// TIA Portal project "openness_project_20230906_002120" (V17)

(* hardware
DEVICE "n0001-zp001-el001-k30001"  S7-1500 station
   slot 0: "Rail_0"  Rack  6ES7 590-1***0-0AA0
   slot 1: "n0001-zp001-el001-k30001"  CPU 1517F-3 PN/DP  6ES7 517-3FP00-0AB0  V2.9
      slot 3: "CPU display_1"  6ES7591-1BA00-0AA0
      slot 32768: "PROFINET interface_1"  X1
         slot 32769: "Port_1"  X1 P1
         slot 32770: "Port_2"  X1 P2
      slot 33024: "PROFINET interface_2"  X2
         slot 33025: "Port_1"  X2 P1
      slot 33280: "DP interface_1"  X3
      slot 34817: "Virtual CP interface port_1"  Virtual CP interface port  Virtual CP interface port
   slot 2: "n0001-zp001-el001-k30002"  CM 1542-1  6GK7 542-1AX00-0XE0  V3.0
DEVICE "n0006-zp001-el001-k25501"  PnPn.Device
   slot 0: "Rack"  Rail  1.0
   slot 0: "n0006-zp001-el001-k25501"  PN/PN Coupler  6ES7 158-3AD10-0XA0  V4.2
   slot 1: "SC01-SORTER-UCOY"  PN/PN Coupler  6ES7 158-3AD10-0XA0  V4.2
   slot 127: "BA 2xRJ45"  BA 2xRJ45  6ES7 193-6AR00-0AA0  V0.0
      slot 1: "Port_1"  X1 P1 R  6ES7 193-6AR00-0AA0  V0.0
      slot 2: "Port_2"  X1 P2 R  6ES7 193-6AR00-0AA0  V0.0
   slot 127: "BA 2xRJ45"  BA 2xRJ45  6ES7 193-6AR00-0AA0  V0.0
      slot 1: "Port_1"  X2 P1 R  6ES7 193-6AR00-0AA0  V0.0
      slot 2: "Port_2"  X2 P2 R  6ES7 193-6AR00-0AA0  V0.0
DEVICE "n0007-zp001-el001-k25502"  PnPn.Device
   slot 0: "Rack"  Rail  1.0
   slot 0: "n0007-zp001-el001-k25502"  PN/PN Coupler  6ES7 158-3AD10-0XA0  V4.2
   slot 1: "SC02-SORTER-LCOY"  PN/PN Coupler  6ES7 158-3AD10-0XA0  V4.2
   slot 127: "BA 2xRJ45"  BA 2xRJ45  6ES7 193-6AR00-0AA0  V0.0
      slot 1: "Port_1"  X1 P1 R  6ES7 193-6AR00-0AA0  V0.0
      slot 2: "Port_2"  X1 P2 R  6ES7 193-6AR00-0AA0  V0.0
   slot 127: "BA 2xRJ45"  BA 2xRJ45  6ES7 193-6AR00-0AA0  V0.0
      slot 1: "Port_1"  X2 P1 R  6ES7 193-6AR00-0AA0  V0.0
      slot 2: "Port_2"  X2 P2 R  6ES7 193-6AR00-0AA0  V0.0
DEVICE "n0008-zp001-el001-k25601"  PnPn.Device
   slot 0: "Rack"  Rail  1.0
   slot 0: "n0008-zp001-el001-k25601"  PN/PN Coupler  6ES7 158-3AD10-0XA0  V4.2
   slot 1: "SF03-SORTER-UFLY"  PN/PN Coupler  6ES7 158-3AD10-0XA0  V4.2
   slot 127: "BA 2xRJ45"  BA 2xRJ45  6ES7 193-6AR00-0AA0  V0.0
      slot 1: "Port_1"  X1 P1 R  6ES7 193-6AR00-0AA0  V0.0
      slot 2: "Port_2"  X1 P2 R  6ES7 193-6AR00-0AA0  V0.0
   slot 127: "BA 2xRJ45"  BA 2xRJ45  6ES7 193-6AR00-0AA0  V0.0
      slot 1: "Port_1"  X2 P1 R  6ES7 193-6AR00-0AA0  V0.0
      slot 2: "Port_2"  X2 P2 R  6ES7 193-6AR00-0AA0  V0.0
DEVICE "n0009-zp001-el001-k25602"  PnPn.Device
   slot 0: "Rack"  Rail  1.0
   slot 0: "n0009-zp001-el001-k25602"  PN/PN Coupler  6ES7 158-3AD10-0XA0  V4.2
   slot 1: "SF04-SORTER-LFLY"  PN/PN Coupler  6ES7 158-3AD10-0XA0  V4.2
   slot 127: "BA 2xRJ45"  BA 2xRJ45  6ES7 193-6AR00-0AA0  V0.0
      slot 1: "Port_1"  X1 P1 R  6ES7 193-6AR00-0AA0  V0.0
      slot 2: "Port_2"  X1 P2 R  6ES7 193-6AR00-0AA0  V0.0
   slot 127: "BA 2xRJ45"  BA 2xRJ45  6ES7 193-6AR00-0AA0  V0.0
      slot 1: "Port_1"  X2 P1 R  6ES7 193-6AR00-0AA0  V0.0
      slot 2: "Port_2"  X2 P2 R  6ES7 193-6AR00-0AA0  V0.0
DEVICE "n0005-zp001-el001-k40001"  ET 200SP-Station
   slot 0: "Rack_0"  Rack  6ES5 710-8MAx1
   slot 0: "n0005-zp001-el001-k40001"  IM 155-6 PN ST  6ES7 155-6AU01-0BN0  V4.2
   slot 1: "-K40002"  DI 16x24VDC ST  6ES7 131-6BH01-0BA0  V0.0
      slot 1: "-K40002"  DI 16x24VDC ST
   slot 2: "-K40003"  DI 16x24VDC ST  6ES7 131-6BH01-0BA0  V0.0
      slot 1: "-K40003"  DI 16x24VDC ST
   slot 3: "-K40004"  DI 16x24VDC ST  6ES7 131-6BH01-0BA0  V0.0
      slot 1: "-K40004"  DI 16x24VDC ST
   slot 4: "-K40005"  DI 16x24VDC ST  6ES7 131-6BH01-0BA0  V0.0
      slot 1: "-K40005"  DI 16x24VDC ST
   slot 5: "-K40006"  DI 16x24VDC ST  6ES7 131-6BH01-0BA0  V0.0
      slot 1: "-K40006"  DI 16x24VDC ST
   slot 6: "-K40007"  DI 16x24VDC ST  6ES7 131-6BH01-0BA0  V0.0
      slot 1: "-K40007"  DI 16x24VDC ST
   slot 7: "-K40008"  DI 16x24VDC ST  6ES7 131-6BH01-0BA0  V0.0
      slot 1: "-K40008"  DI 16x24VDC ST
   slot 8: "-K40009"  DI 16x24VDC ST  6ES7 131-6BH01-0BA0  V0.0
      slot 1: "-K40009"  DI 16x24VDC ST
   slot 9: "-K40010"  DI 16x24VDC ST  6ES7 131-6BH01-0BA0  V0.0
      slot 1: "-K40010"  DI 16x24VDC ST
   slot 10: "-K40011"  DI 16x24VDC ST  6ES7 131-6BH01-0BA0  V0.0
      slot 1: "-K40011"  DI 16x24VDC ST
   slot 11: "-K40012"  DI 16x24VDC ST  6ES7 131-6BH01-0BA0  V0.0
      slot 1: "-K40012"  DI 16x24VDC ST
   slot 12: "-K40013"  DI 16x24VDC ST  6ES7 131-6BH01-0BA0  V0.0
      slot 1: "-K40013"  DI 16x24VDC ST
   slot 13: "-K40014"  DI 16x24VDC ST  6ES7 131-6BH01-0BA0  V0.0
      slot 1: "-K40014"  DI 16x24VDC ST
   slot 14: "-K40015"  DI 16x24VDC ST  6ES7 131-6BH01-0BA0  V0.0
      slot 1: "-K40015"  DI 16x24VDC ST
   slot 15: "-K40016"  DI 16x24VDC ST  6ES7 131-6BH01-0BA0  V0.0
      slot 1: "-K40016"  DI 16x24VDC ST
   slot 16: "-K40017"  DI 16x24VDC ST  6ES7 131-6BH01-0BA0  V0.0
      slot 1: "-K40017"  DI 16x24VDC ST
   slot 17: "-K40018"  DI 16x24VDC ST  6ES7 131-6BH01-0BA0  V0.0
      slot 1: "-K40018"  DI 16x24VDC ST
   slot 18: "-K40019"  F-DI 8x24VDC HF  6ES7 136-6BA00-0CA0  V1.0
      slot 1: "-K40019"  F-DI 8x24VDC HF
   slot 19: "-K40020"  DQ 16x24VDC/0.5A ST  6ES7 132-6BH01-0BA0  V0.0
      slot 1: "-K40020"  DQ 16x24VDC/0.5A ST
   slot 20: "Server module_1"  Server module  6ES7 193-6PA00-0AA0  V1.1
      slot 1: "Server module_1"  Server module
   slot 127: "BA 2xRJ45"  BA 2xRJ45  6ES7 193-6AR00-0AA0  V0.0
      slot 1: "Port_1"  X1 P1 R  6ES7 193-6AR00-0AA0  V0.0
      slot 2: "Port_2"  X1 P2 R  6ES7 193-6AR00-0AA0  V0.0
DEVICE "n0013-uf317-xn10"  GSD.Device.PN
   slot 0: "Rack"  Rack  V1.0
   slot 0: "n0013-uf317-xn10"  55556 MVK-MPNIO F DI16/8  55556
      slot 0: "55556 MVK-MPNIO F DI16/8_1"  55556 MVK-MPNIO F DI16/8
      slot 1: "55556 MVK-MPNIO F DI16/8"  55556 MVK-MPNIO F DI16/8
         slot 1: "Port 1"  Port 1
         slot 2: "Port 2"  Port 2
      slot 1: "Power module_1"  Power module
         slot 0: "Power module"  Power module
   slot 2: "-XN10"  FS Data
      slot 0: "-XN10"  FS Data
DEVICE "n0015-uc16-el001-k30001"  ET 200SP-Station
   slot 0: "Rack_0"  Rack  6ES5 710-8MAx1
   slot 0: "n0015-uc16-el001-k30001"  IM 155-6 PN ST  6ES7 155-6AU01-0BN0  V4.2
   slot 1: "-K30002"  DI 16x24VDC ST  6ES7 131-6BH01-0BA0  V0.0
      slot 1: "-K30002"  DI 16x24VDC ST
   slot 2: "-K30003"  DI 16x24VDC ST  6ES7 131-6BH01-0BA0  V0.0
      slot 1: "-K30003"  DI 16x24VDC ST
   slot 3: "-K30004"  F-DI 8x24VDC HF  6ES7 136-6BA00-0CA0  V1.0
      slot 1: "-K30004"  F-DI 8x24VDC HF
   slot 4: "-K30005"  F-DI 8x24VDC HF  6ES7 136-6BA00-0CA0  V1.0
      slot 1: "-K30005"  F-DI 8x24VDC HF
   slot 5: "-K30006"  F-DI 8x24VDC HF  6ES7 136-6BA00-0CA0  V1.0
      slot 1: "-K30006"  F-DI 8x24VDC HF
   slot 6: "-K30007"  F-DI 8x24VDC HF  6ES7 136-6BA00-0CA0  V1.0
      slot 1: "-K30007"  F-DI 8x24VDC HF
   slot 7: "-K30008"  F-DQ 4x24VDC/2A PM HF  6ES7 136-6DB00-0CA0  V2.0
      slot 1: "-K30008"  F-DQ 4x24VDC/2A PM HF
   slot 8: "-K30009"  F-DQ 4x24VDC/2A PM HF  6ES7 136-6DB00-0CA0  V2.0
      slot 1: "-K30009"  F-DQ 4x24VDC/2A PM HF
   slot 9: "-K30010"  F-DQ 4x24VDC/2A PM HF  6ES7 136-6DB00-0CA0  V2.0
      slot 1: "-K30010"  F-DQ 4x24VDC/2A PM HF
   slot 10: "-K30011"  F-DQ 4x24VDC/2A PM HF  6ES7 136-6DB00-0CA0  V2.0
      slot 1: "-K30011"  F-DQ 4x24VDC/2A PM HF
   slot 11: "-K30012"  F-DQ 4x24VDC/2A PM HF  6ES7 136-6DB00-0CA0  V2.0
      slot 1: "-K30012"  F-DQ 4x24VDC/2A PM HF
   slot 12: "-K30013"  F-DQ 4x24VDC/2A PM HF  6ES7 136-6DB00-0CA0  V2.0
      slot 1: "-K30013"  F-DQ 4x24VDC/2A PM HF
   slot 13: "Server module_1"  Server module  6ES7 193-6PA00-0AA0  V1.1
      slot 1: "Server module_1"  Server module
   slot 127: "BA 2xRJ45"  BA 2xRJ45  6ES7 193-6AR00-0AA0  V0.0
      slot 1: "Port_1"  X1 P1 R  6ES7 193-6AR00-0AA0  V0.0
      slot 2: "Port_2"  X1 P2 R  6ES7 193-6AR00-0AA0  V0.0
DEVICE "n0016-uc164-xn10"  GSD.Device.PN
   slot 0: "Rack"  Rack  V1.0
   slot 0: "n0016-uc164-xn10"  55556 MVK-MPNIO F DI16/8  55556
      slot 0: "55556 MVK-MPNIO F DI16/8_1"  55556 MVK-MPNIO F DI16/8
      slot 1: "55556 MVK-MPNIO F DI16/8"  55556 MVK-MPNIO F DI16/8
         slot 1: "Port 1"  Port 1
         slot 2: "Port 2"  Port 2
      slot 1: "Power module_1"  Power module
         slot 0: "Power module"  Power module
   slot 2: "-XN10"  FS Data
      slot 0: "-XN10"  FS Data
DEVICE "n0017-lv004-el001-k30001"  ET 200SP-Station
   slot 0: "Rack_0"  Rack  6ES5 710-8MAx1
   slot 0: "n0017-lv004-el001-k30001"  IM 155-6 PN ST  6ES7 155-6AU01-0BN0  V4.2
   slot 1: "-K30002"  DI 16x24VDC ST  6ES7 131-6BH01-0BA0  V0.0
      slot 1: "-K30002"  DI 16x24VDC ST
   slot 2: "-K30003"  F-DI 8x24VDC HF  6ES7 136-6BA00-0CA0  V1.0
      slot 1: "-K30003"  F-DI 8x24VDC HF
   slot 3: "-K30004"  F-DI 8x24VDC HF  6ES7 136-6BA00-0CA0  V1.0
      slot 1: "-K30004"  F-DI 8x24VDC HF
   slot 4: "-K30005"  F-DQ 4x24VDC/2A PM HF  6ES7 136-6DB00-0CA0  V2.0
      slot 1: "-K30005"  F-DQ 4x24VDC/2A PM HF
   slot 5: "-K30006"  F-DQ 4x24VDC/2A PM HF  6ES7 136-6DB00-0CA0  V2.0
      slot 1: "-K30006"  F-DQ 4x24VDC/2A PM HF
   slot 6: "Server module_1"  Server module  6ES7 193-6PA00-0AA0  V1.1
      slot 1: "Server module_1"  Server module
   slot 127: "BA 2xRJ45"  BA 2xRJ45  6ES7 193-6AR00-0AA0  V0.0
      slot 1: "Port_1"  X1 P1 R  6ES7 193-6AR00-0AA0  V0.0
      slot 2: "Port_2"  X1 P2 R  6ES7 193-6AR00-0AA0  V0.0
DEVICE "n0018-lv004-el001-k30001"  ET 200SP-Station
   slot 0: "Rack_0"  Rack  6ES5 710-8MAx1
   slot 0: "n0018-lv004-el001-k30001"  IM 155-6 PN ST  6ES7 155-6AU01-0BN0  V4.2
   slot 1: "-K30002"  DI 16x24VDC ST  6ES7 131-6BH01-0BA0  V0.0
      slot 1: "-K30002"  DI 16x24VDC ST
   slot 2: "-K30003"  F-DI 8x24VDC HF  6ES7 136-6BA00-0CA0  V1.0
      slot 1: "-K30003"  F-DI 8x24VDC HF
   slot 3: "-K30004"  F-DI 8x24VDC HF  6ES7 136-6BA00-0CA0  V1.0
      slot 1: "-K30004"  F-DI 8x24VDC HF
   slot 4: "-K30005"  F-DQ 4x24VDC/2A PM HF  6ES7 136-6DB00-0CA0  V2.0
      slot 1: "-K30005"  F-DQ 4x24VDC/2A PM HF
   slot 5: "-K30006"  F-DQ 4x24VDC/2A PM HF  6ES7 136-6DB00-0CA0  V2.0
      slot 1: "-K30006"  F-DQ 4x24VDC/2A PM HF
   slot 6: "Server module_1"  Server module  6ES7 193-6PA00-0AA0  V1.1
      slot 1: "Server module_1"  Server module
   slot 127: "BA 2xRJ45"  BA 2xRJ45  6ES7 193-6AR00-0AA0  V0.0
      slot 1: "Port_1"  X1 P1 R  6ES7 193-6AR00-0AA0  V0.0
      slot 2: "Port_2"  X1 P2 R  6ES7 193-6AR00-0AA0  V0.0
DEVICE "n0020-uc15-el001-k30001"  ET 200SP-Station
   slot 0: "Rack_0"  Rack  6ES5 710-8MAx1
   slot 0: "n0020-uc15-el001-k30001"  IM 155-6 PN ST  6ES7 155-6AU01-0BN0  V4.2
   slot 1: "-K30002"  DI 16x24VDC ST  6ES7 131-6BH01-0BA0  V0.0
      slot 1: "-K30002"  DI 16x24VDC ST
   slot 2: "-K30003"  DI 16x24VDC ST  6ES7 131-6BH01-0BA0  V0.0
      slot 1: "-K30003"  DI 16x24VDC ST
   slot 3: "-K30004"  F-DI 8x24VDC HF  6ES7 136-6BA00-0CA0  V1.0
      slot 1: "-K30004"  F-DI 8x24VDC HF
   slot 4: "-K30005"  F-DI 8x24VDC HF  6ES7 136-6BA00-0CA0  V1.0
      slot 1: "-K30005"  F-DI 8x24VDC HF
   slot 5: "-K30006"  F-DI 8x24VDC HF  6ES7 136-6BA00-0CA0  V1.0
      slot 1: "-K30006"  F-DI 8x24VDC HF
   slot 6: "-K30007"  F-DI 8x24VDC HF  6ES7 136-6BA00-0CA0  V1.0
      slot 1: "-K30007"  F-DI 8x24VDC HF
   slot 7: "-K30008"  F-DQ 4x24VDC/2A PM HF  6ES7 136-6DB00-0CA0  V2.0
      slot 1: "-K30008"  F-DQ 4x24VDC/2A PM HF
   slot 8: "-K30009"  F-DQ 4x24VDC/2A PM HF  6ES7 136-6DB00-0CA0  V2.0
      slot 1: "-K30009"  F-DQ 4x24VDC/2A PM HF
   slot 9: "-K30010"  F-DQ 4x24VDC/2A PM HF  6ES7 136-6DB00-0CA0  V2.0
      slot 1: "-K30010"  F-DQ 4x24VDC/2A PM HF
   slot 10: "-K30011"  F-DQ 4x24VDC/2A PM HF  6ES7 136-6DB00-0CA0  V2.0
      slot 1: "-K30011"  F-DQ 4x24VDC/2A PM HF
   slot 11: "-K30012"  F-DQ 4x24VDC/2A PM HF  6ES7 136-6DB00-0CA0  V2.0
      slot 1: "-K30012"  F-DQ 4x24VDC/2A PM HF
   slot 12: "-K30013"  F-DQ 4x24VDC/2A PM HF  6ES7 136-6DB00-0CA0  V2.0
      slot 1: "-K30013"  F-DQ 4x24VDC/2A PM HF
   slot 13: "Server module_1"  Server module  6ES7 193-6PA00-0AA0  V1.1
      slot 1: "Server module_1"  Server module
   slot 127: "BA 2xRJ45"  BA 2xRJ45  6ES7 193-6AR00-0AA0  V0.0
      slot 1: "Port_1"  X1 P1 R  6ES7 193-6AR00-0AA0  V0.0
      slot 2: "Port_2"  X1 P2 R  6ES7 193-6AR00-0AA0  V0.0
DEVICE "n0023-uc154-xn10"  GSD.Device.PN
   slot 0: "Rack"  Rack  V1.0
   slot 0: "n0023-uc154-xn10"  55556 MVK-MPNIO F DI16/8  55556
      slot 0: "55556 MVK-MPNIO F DI16/8_1"  55556 MVK-MPNIO F DI16/8
      slot 1: "55556 MVK-MPNIO F DI16/8"  55556 MVK-MPNIO F DI16/8
         slot 1: "Port 1"  Port 1
         slot 2: "Port 2"  Port 2
      slot 1: "Power module_1"  Power module
         slot 0: "Power module"  Power module
   slot 2: "-XN10"  FS Data
      slot 0: "-XN10"  FS Data
DEVICE "n0021-icg11-el001-k30001"  ET 200SP-Station
   slot 0: "Rack_0"  Rack  6ES5 710-8MAx1
   slot 0: "n0021-icg11-el001-k30001"  IM 155-6 PN ST  6ES7 155-6AU01-0BN0  V4.2
   slot 1: "-K30002"  DI 16x24VDC ST  6ES7 131-6BH01-0BA0  V0.0
      slot 1: "-K30002"  DI 16x24VDC ST
   slot 2: "-K30003"  F-DI 8x24VDC HF  6ES7 136-6BA00-0CA0  V1.0
      slot 1: "-K30003"  F-DI 8x24VDC HF
   slot 3: "-K30004"  F-DI 8x24VDC HF  6ES7 136-6BA00-0CA0  V1.0
      slot 1: "-K30004"  F-DI 8x24VDC HF
   slot 4: "-K30005"  F-DI 8x24VDC HF  6ES7 136-6BA00-0CA0  V1.0
      slot 1: "-K30005"  F-DI 8x24VDC HF
   slot 5: "-K30006"  F-DI 8x24VDC HF  6ES7 136-6BA00-0CA0  V1.0
      slot 1: "-K30006"  F-DI 8x24VDC HF
   slot 6: "-K30007"  F-DQ 4x24VDC/2A PM HF  6ES7 136-6DB00-0CA0  V2.0
      slot 1: "-K30007"  F-DQ 4x24VDC/2A PM HF
   slot 7: "-K30008"  F-DQ 4x24VDC/2A PM HF  6ES7 136-6DB00-0CA0  V2.0
      slot 1: "-K30008"  F-DQ 4x24VDC/2A PM HF
   slot 8: "-K30009"  F-DQ 4x24VDC/2A PM HF  6ES7 136-6DB00-0CA0  V2.0
      slot 1: "-K30009"  F-DQ 4x24VDC/2A PM HF
   slot 9: "Server module_1"  Server module  6ES7 193-6PA00-0AA0  V1.1
      slot 1: "Server module_1"  Server module
   slot 127: "BA 2xRJ45"  BA 2xRJ45  6ES7 193-6AR00-0AA0  V0.0
      slot 1: "Port_1"  X1 P1 R  6ES7 193-6AR00-0AA0  V0.0
      slot 2: "Port_2"  X1 P2 R  6ES7 193-6AR00-0AA0  V0.0
DEVICE "n0022-icg21-el001-k30001"  ET 200SP-Station
   slot 0: "Rack_0"  Rack  6ES5 710-8MAx1
   slot 0: "n0022-icg21-el001-k30001"  IM 155-6 PN ST  6ES7 155-6AU01-0BN0  V4.2
   slot 1: "-K30002"  DI 16x24VDC ST  6ES7 131-6BH01-0BA0  V0.0
      slot 1: "-K30002"  DI 16x24VDC ST
   slot 2: "-K30003"  F-DI 8x24VDC HF  6ES7 136-6BA00-0CA0  V1.0
      slot 1: "-K30003"  F-DI 8x24VDC HF
   slot 3: "-K30004"  F-DI 8x24VDC HF  6ES7 136-6BA00-0CA0  V1.0
      slot 1: "-K30004"  F-DI 8x24VDC HF
   slot 4: "-K30005"  F-DI 8x24VDC HF  6ES7 136-6BA00-0CA0  V1.0
      slot 1: "-K30005"  F-DI 8x24VDC HF
   slot 5: "-K30006"  F-DI 8x24VDC HF  6ES7 136-6BA00-0CA0  V1.0
      slot 1: "-K30006"  F-DI 8x24VDC HF
   slot 6: "-K30007"  F-DQ 4x24VDC/2A PM HF  6ES7 136-6DB00-0CA0  V2.0
      slot 1: "-K30007"  F-DQ 4x24VDC/2A PM HF
   slot 7: "-K30008"  F-DQ 4x24VDC/2A PM HF  6ES7 136-6DB00-0CA0  V2.0
      slot 1: "-K30008"  F-DQ 4x24VDC/2A PM HF
   slot 8: "-K30009"  F-DQ 4x24VDC/2A PM HF  6ES7 136-6DB00-0CA0  V2.0
      slot 1: "-K30009"  F-DQ 4x24VDC/2A PM HF
   slot 9: "Server module_1"  Server module  6ES7 193-6PA00-0AA0  V1.1
      slot 1: "Server module_1"  Server module
   slot 127: "BA 2xRJ45"  BA 2xRJ45  6ES7 193-6AR00-0AA0  V0.0
      slot 1: "Port_1"  X1 P1 R  6ES7 193-6AR00-0AA0  V0.0
      slot 2: "Port_2"  X1 P2 R  6ES7 193-6AR00-0AA0  V0.0
DEVICE "n0025-uc14-el001-k30001"  ET 200SP-Station
   slot 0: "Rack_0"  Rack  6ES5 710-8MAx1
   slot 0: "n0025-uc14-el001-k30001"  IM 155-6 PN ST  6ES7 155-6AU01-0BN0  V4.2
   slot 1: "-K30002"  DI 16x24VDC ST  6ES7 131-6BH01-0BA0  V0.0
      slot 1: "-K30002"  DI 16x24VDC ST
   slot 2: "-K30003"  DI 16x24VDC ST  6ES7 131-6BH01-0BA0  V0.0
      slot 1: "-K30003"  DI 16x24VDC ST
   slot 3: "-K30004"  F-DI 8x24VDC HF  6ES7 136-6BA00-0CA0  V1.0
      slot 1: "-K30004"  F-DI 8x24VDC HF
   slot 4: "-K30005"  F-DI 8x24VDC HF  6ES7 136-6BA00-0CA0  V1.0
      slot 1: "-K30005"  F-DI 8x24VDC HF
   slot 5: "-K30006"  F-DI 8x24VDC HF  6ES7 136-6BA00-0CA0  V1.0
      slot 1: "-K30006"  F-DI 8x24VDC HF
   slot 6: "-K30007"  F-DI 8x24VDC HF  6ES7 136-6BA00-0CA0  V1.0
      slot 1: "-K30007"  F-DI 8x24VDC HF
   slot 7: "-K30008"  F-DQ 4x24VDC/2A PM HF  6ES7 136-6DB00-0CA0  V2.0
      slot 1: "-K30008"  F-DQ 4x24VDC/2A PM HF
   slot 8: "-K30009"  F-DQ 4x24VDC/2A PM HF  6ES7 136-6DB00-0CA0  V2.0
      slot 1: "-K30009"  F-DQ 4x24VDC/2A PM HF
   slot 9: "-K30010"  F-DQ 4x24VDC/2A PM HF  6ES7 136-6DB00-0CA0  V2.0
      slot 1: "-K30010"  F-DQ 4x24VDC/2A PM HF
   slot 10: "-K30011"  F-DQ 4x24VDC/2A PM HF  6ES7 136-6DB00-0CA0  V2.0
      slot 1: "-K30011"  F-DQ 4x24VDC/2A PM HF
   slot 11: "-K30012"  F-DQ 4x24VDC/2A PM HF  6ES7 136-6DB00-0CA0  V2.0
      slot 1: "-K30012"  F-DQ 4x24VDC/2A PM HF
   slot 12: "-K30013"  F-DQ 4x24VDC/2A PM HF  6ES7 136-6DB00-0CA0  V2.0
      slot 1: "-K30013"  F-DQ 4x24VDC/2A PM HF
   slot 13: "Server module_1"  Server module  6ES7 193-6PA00-0AA0  V1.1
      slot 1: "Server module_1"  Server module
   slot 127: "BA 2xRJ45"  BA 2xRJ45  6ES7 193-6AR00-0AA0  V0.0
      slot 1: "Port_1"  X1 P1 R  6ES7 193-6AR00-0AA0  V0.0
      slot 2: "Port_2"  X1 P2 R  6ES7 193-6AR00-0AA0  V0.0
DEVICE "n0026-uc144-xn10"  GSD.Device.PN
   slot 0: "Rack"  Rack  V1.0
   slot 0: "n0026-uc144-xn10"  55556 MVK-MPNIO F DI16/8  55556
      slot 0: "55556 MVK-MPNIO F DI16/8_1"  55556 MVK-MPNIO F DI16/8
      slot 1: "55556 MVK-MPNIO F DI16/8"  55556 MVK-MPNIO F DI16/8
         slot 1: "Port 1"  Port 1
         slot 2: "Port 2"  Port 2
      slot 1: "Power module_1"  Power module
         slot 0: "Power module"  Power module
   slot 2: "-XN10"  FS Data
      slot 0: "-XN10"  FS Data
DEVICE "n0038-uc1-el001-k30001"  ET 200SP-Station
   slot 0: "Rack_0"  Rack  6ES5 710-8MAx1
   slot 0: "n0038-uc1-el001-k30001"  IM 155-6 PN ST  6ES7 155-6AU01-0BN0  V4.2
   slot 1: "-K30002"  DI 16x24VDC ST  6ES7 131-6BH01-0BA0  V0.0
      slot 1: "-K30002"  DI 16x24VDC ST
   slot 2: "-K30003"  F-DI 8x24VDC HF  6ES7 136-6BA00-0CA0  V1.0
      slot 1: "-K30003"  F-DI 8x24VDC HF
   slot 3: "-K30004"  F-DI 8x24VDC HF  6ES7 136-6BA00-0CA0  V1.0
      slot 1: "-K30004"  F-DI 8x24VDC HF
   slot 4: "-K30005"  F-DQ 4x24VDC/2A PM HF  6ES7 136-6DB00-0CA0  V2.0
      slot 1: "-K30005"  F-DQ 4x24VDC/2A PM HF
   slot 5: "-K30006"  DQ 16x24VDC/0.5A ST  6ES7 132-6BH01-0BA0  V0.0
      slot 1: "-K30006"  DQ 16x24VDC/0.5A ST
   slot 6: "Server module_1"  Server module  6ES7 193-6PA00-0AA0  V1.1
      slot 1: "Server module_1"  Server module
   slot 127: "BA 2xRJ45"  BA 2xRJ45  6ES7 193-6AR00-0AA0  V0.0
      slot 1: "Port_1"  X1 P1 R  6ES7 193-6AR00-0AA0  V0.0
      slot 2: "Port_2"  X1 P2 R  6ES7 193-6AR00-0AA0  V0.0
DEVICE "n0039-lv001-el001-k30001"  ET 200SP-Station
   slot 0: "Rack_0"  Rack  6ES5 710-8MAx1
   slot 0: "n0039-lv001-el001-k30001"  IM 155-6 PN ST  6ES7 155-6AU01-0BN0  V4.2
   slot 1: "-K30002"  DI 16x24VDC ST  6ES7 131-6BH01-0BA0  V0.0
      slot 1: "-K30002"  DI 16x24VDC ST
   slot 2: "-K30003"  F-DI 8x24VDC HF  6ES7 136-6BA00-0CA0  V1.0
      slot 1: "-K30003"  F-DI 8x24VDC HF
   slot 3: "-K30004"  F-DQ 4x24VDC/2A PM HF  6ES7 136-6DB00-0CA0  V2.0
      slot 1: "-K30004"  F-DQ 4x24VDC/2A PM HF
   slot 4: "Server module_1"  Server module  6ES7 193-6PA00-0AA0  V1.1
      slot 1: "Server module_1"  Server module
   slot 127: "BA 2xRJ45"  BA 2xRJ45  6ES7 193-6AR00-0AA0  V0.0
      slot 1: "Port_1"  X1 P1 R  6ES7 193-6AR00-0AA0  V0.0
      slot 2: "Port_2"  X1 P2 R  6ES7 193-6AR00-0AA0  V0.0
DEVICE "n0040-lv001-el001-k30001"  ET 200SP-Station
   slot 0: "Rack_0"  Rack  6ES5 710-8MAx1
   slot 0: "n0040-lv001-el001-k30001"  IM 155-6 PN ST  6ES7 155-6AU01-0BN0  V4.2
   slot 1: "-K30002"  DI 16x24VDC ST  6ES7 131-6BH01-0BA0  V0.0
      slot 1: "-K30002"  DI 16x24VDC ST
   slot 2: "-K30003"  F-DI 8x24VDC HF  6ES7 136-6BA00-0CA0  V1.0
      slot 1: "-K30003"  F-DI 8x24VDC HF
   slot 3: "-K30004"  F-DQ 4x24VDC/2A PM HF  6ES7 136-6DB00-0CA0  V2.0
      slot 1: "-K30004"  F-DQ 4x24VDC/2A PM HF
   slot 4: "Server module_1"  Server module  6ES7 193-6PA00-0AA0  V1.1
      slot 1: "Server module_1"  Server module
   slot 127: "BA 2xRJ45"  BA 2xRJ45  6ES7 193-6AR00-0AA0  V0.0
      slot 1: "Port_1"  X1 P1 R  6ES7 193-6AR00-0AA0  V0.0
      slot 2: "Port_2"  X1 P2 R  6ES7 193-6AR00-0AA0  V0.0
DEVICE "n0041-uf31-el002-k30001"  ET 200SP-Station
   slot 0: "Rack_0"  Rack  6ES5 710-8MAx1
   slot 0: "n0041-uf31-el002-k30001"  IM 155-6 PN ST  6ES7 155-6AU01-0BN0  V4.2
   slot 1: "-K30002"  DI 16x24VDC ST  6ES7 131-6BH01-0BA0  V0.0
      slot 1: "-K30002"  DI 16x24VDC ST
   slot 2: "-K30003"  F-DI 8x24VDC HF  6ES7 136-6BA00-0CA0  V1.0
      slot 1: "-K30003"  F-DI 8x24VDC HF
   slot 3: "-K30004"  F-DI 8x24VDC HF  6ES7 136-6BA00-0CA0  V1.0
      slot 1: "-K30004"  F-DI 8x24VDC HF
   slot 4: "-K30005"  F-DQ 4x24VDC/2A PM HF  6ES7 136-6DB00-0CA0  V2.0
      slot 1: "-K30005"  F-DQ 4x24VDC/2A PM HF
   slot 5: "Server module_1"  Server module  6ES7 193-6PA00-0AA0  V1.1
      slot 1: "Server module_1"  Server module
   slot 127: "BA 2xRJ45"  BA 2xRJ45  6ES7 193-6AR00-0AA0  V0.0
      slot 1: "Port_1"  X1 P1 R  6ES7 193-6AR00-0AA0  V0.0
      slot 2: "Port_2"  X1 P2 R  6ES7 193-6AR00-0AA0  V0.0
DEVICE "n0042-uf41-el002-k30001"  ET 200SP-Station
   slot 0: "Rack_0"  Rack  6ES5 710-8MAx1
   slot 0: "n0042-uf41-el002-k30001"  IM 155-6 PN ST  6ES7 155-6AU01-0BN0  V4.2
   slot 1: "-K30002"  DI 16x24VDC ST  6ES7 131-6BH01-0BA0  V0.0
      slot 1: "-K30002"  DI 16x24VDC ST
   slot 2: "-K30003"  F-DI 8x24VDC HF  6ES7 136-6BA00-0CA0  V1.0
      slot 1: "-K30003"  F-DI 8x24VDC HF
   slot 3: "-K30004"  F-DQ 4x24VDC/2A PM HF  6ES7 136-6DB00-0CA0  V2.0
      slot 1: "-K30004"  F-DQ 4x24VDC/2A PM HF
   slot 4: "-K30005"  F-DQ 4x24VDC/2A PM HF  6ES7 136-6DB00-0CA0  V2.0
      slot 1: "-K30005"  F-DQ 4x24VDC/2A PM HF
   slot 5: "Server module_1"  Server module  6ES7 193-6PA00-0AA0  V1.1
      slot 1: "Server module_1"  Server module
   slot 127: "BA 2xRJ45"  BA 2xRJ45  6ES7 193-6AR00-0AA0  V0.0
      slot 1: "Port_1"  X1 P1 R  6ES7 193-6AR00-0AA0  V0.0
      slot 2: "Port_2"  X1 P2 R  6ES7 193-6AR00-0AA0  V0.0
DEVICE "n0044-ct1-el001-k30001"  ET 200SP-Station
   slot 0: "Rack_0"  Rack  6ES5 710-8MAx1
   slot 0: "n0044-ct1-el001-k30001"  IM 155-6 PN ST  6ES7 155-6AU01-0BN0  V4.2
   slot 1: "-K30002"  DI 16x24VDC ST  6ES7 131-6BH01-0BA0  V0.0
      slot 1: "-K30002"  DI 16x24VDC ST
   slot 2: "-K30003"  F-DI 8x24VDC HF  6ES7 136-6BA00-0CA0  V1.0
      slot 1: "-K30003"  F-DI 8x24VDC HF
   slot 3: "-K30004"  F-DI 8x24VDC HF  6ES7 136-6BA00-0CA0  V1.0
      slot 1: "-K30004"  F-DI 8x24VDC HF
   slot 4: "-K30005"  F-DI 8x24VDC HF  6ES7 136-6BA00-0CA0  V1.0
      slot 1: "-K30005"  F-DI 8x24VDC HF
   slot 5: "-K30006"  F-DI 8x24VDC HF  6ES7 136-6BA00-0CA0  V1.0
      slot 1: "-K30006"  F-DI 8x24VDC HF
   slot 6: "-K30007"  F-DI 8x24VDC HF  6ES7 136-6BA00-0CA0  V1.0
      slot 1: "-K30007"  F-DI 8x24VDC HF
   slot 7: "-K30008"  F-DQ 4x24VDC/2A PM HF  6ES7 136-6DB00-0CA0  V2.0
      slot 1: "-K30008"  F-DQ 4x24VDC/2A PM HF
   slot 8: "-K30009"  F-DQ 4x24VDC/2A PM HF  6ES7 136-6DB00-0CA0  V2.0
      slot 1: "-K30009"  F-DQ 4x24VDC/2A PM HF
   slot 9: "Server module_1"  Server module  6ES7 193-6PA00-0AA0  V1.1
      slot 1: "Server module_1"  Server module
   slot 127: "BA 2xRJ45"  BA 2xRJ45  6ES7 193-6AR00-0AA0  V0.0
      slot 1: "Port_1"  X1 P1 R  6ES7 193-6AR00-0AA0  V0.0
      slot 2: "Port_2"  X1 P2 R  6ES7 193-6AR00-0AA0  V0.0
DEVICE "n0045-ct1-el002-k30001"  ET 200SP-Station
   slot 0: "Rack_0"  Rack  6ES5 710-8MAx1
   slot 0: "n0045-ct1-el002-k30001"  IM 155-6 PN ST  6ES7 155-6AU01-0BN0  V4.2
   slot 1: "-K30002"  DI 16x24VDC ST  6ES7 131-6BH01-0BA0  V0.0
      slot 1: "-K30002"  DI 16x24VDC ST
   slot 2: "-K30003"  F-DI 8x24VDC HF  6ES7 136-6BA00-0CA0  V1.0
      slot 1: "-K30003"  F-DI 8x24VDC HF
   slot 3: "-K30004"  F-DI 8x24VDC HF  6ES7 136-6BA00-0CA0  V1.0
      slot 1: "-K30004"  F-DI 8x24VDC HF
   slot 4: "-K30005"  F-DI 8x24VDC HF  6ES7 136-6BA00-0CA0  V1.0
      slot 1: "-K30005"  F-DI 8x24VDC HF
   slot 5: "-K30006"  F-DI 8x24VDC HF  6ES7 136-6BA00-0CA0  V1.0
      slot 1: "-K30006"  F-DI 8x24VDC HF
   slot 6: "-K30007"  F-DI 8x24VDC HF  6ES7 136-6BA00-0CA0  V1.0
      slot 1: "-K30007"  F-DI 8x24VDC HF
   slot 7: "-K30008"  F-DQ 4x24VDC/2A PM HF  6ES7 136-6DB00-0CA0  V2.0
      slot 1: "-K30008"  F-DQ 4x24VDC/2A PM HF
   slot 8: "-K30009"  F-DQ 4x24VDC/2A PM HF  6ES7 136-6DB00-0CA0  V2.0
      slot 1: "-K30009"  F-DQ 4x24VDC/2A PM HF
   slot 9: "Server module_1"  Server module  6ES7 193-6PA00-0AA0  V1.1
      slot 1: "Server module_1"  Server module
   slot 127: "BA 2xRJ45"  BA 2xRJ45  6ES7 193-6AR00-0AA0  V0.0
      slot 1: "Port_1"  X1 P1 R  6ES7 193-6AR00-0AA0  V0.0
      slot 2: "Port_2"  X1 P2 R  6ES7 193-6AR00-0AA0  V0.0
DEVICE "n0046-ct1-el003-k30001"  ET 200SP-Station
   slot 0: "Rack_0"  Rack  6ES5 710-8MAx1
   slot 0: "n0046-ct1-el003-k30001"  IM 155-6 PN ST  6ES7 155-6AU01-0BN0  V4.2
   slot 1: "-K30002"  DI 16x24VDC ST  6ES7 131-6BH01-0BA0  V0.0
      slot 1: "-K30002"  DI 16x24VDC ST
   slot 2: "-K30003"  F-DI 8x24VDC HF  6ES7 136-6BA00-0CA0  V1.0
      slot 1: "-K30003"  F-DI 8x24VDC HF
   slot 3: "-K30004"  F-DI 8x24VDC HF  6ES7 136-6BA00-0CA0  V1.0
      slot 1: "-K30004"  F-DI 8x24VDC HF
   slot 4: "-K30005"  F-DI 8x24VDC HF  6ES7 136-6BA00-0CA0  V1.0
      slot 1: "-K30005"  F-DI 8x24VDC HF
   slot 5: "-K30006"  F-DI 8x24VDC HF  6ES7 136-6BA00-0CA0  V1.0
      slot 1: "-K30006"  F-DI 8x24VDC HF
   slot 6: "-K30007"  F-DI 8x24VDC HF  6ES7 136-6BA00-0CA0  V1.0
      slot 1: "-K30007"  F-DI 8x24VDC HF
   slot 7: "-K30008"  F-DQ 4x24VDC/2A PM HF  6ES7 136-6DB00-0CA0  V2.0
      slot 1: "-K30008"  F-DQ 4x24VDC/2A PM HF
   slot 8: "-K30009"  F-DQ 4x24VDC/2A PM HF  6ES7 136-6DB00-0CA0  V2.0
      slot 1: "-K30009"  F-DQ 4x24VDC/2A PM HF
   slot 9: "Server module_1"  Server module  6ES7 193-6PA00-0AA0  V1.1
      slot 1: "Server module_1"  Server module
   slot 127: "BA 2xRJ45"  BA 2xRJ45  6ES7 193-6AR00-0AA0  V0.0
      slot 1: "Port_1"  X1 P1 R  6ES7 193-6AR00-0AA0  V0.0
      slot 2: "Port_2"  X1 P2 R  6ES7 193-6AR00-0AA0  V0.0
DEVICE "n0047-lv002-el001-k30001"  ET 200SP-Station
   slot 0: "Rack_0"  Rack  6ES5 710-8MAx1
   slot 0: "n0047-lv002-el001-k30001"  IM 155-6 PN ST  6ES7 155-6AU01-0BN0  V4.2
   slot 1: "-K30002"  DI 16x24VDC ST  6ES7 131-6BH01-0BA0  V0.0
      slot 1: "-K30002"  DI 16x24VDC ST
   slot 2: "-K30003"  F-DI 8x24VDC HF  6ES7 136-6BA00-0CA0  V1.0
      slot 1: "-K30003"  F-DI 8x24VDC HF
   slot 3: "-K30004"  F-DQ 4x24VDC/2A PM HF  6ES7 136-6DB00-0CA0  V2.0
      slot 1: "-K30004"  F-DQ 4x24VDC/2A PM HF
   slot 4: "Server module_1"  Server module  6ES7 193-6PA00-0AA0  V1.1
      slot 1: "Server module_1"  Server module
   slot 127: "BA 2xRJ45"  BA 2xRJ45  6ES7 193-6AR00-0AA0  V0.0
      slot 1: "Port_1"  X1 P1 R  6ES7 193-6AR00-0AA0  V0.0
      slot 2: "Port_2"  X1 P2 R  6ES7 193-6AR00-0AA0  V0.0
DEVICE "n0048-lv002-el001-k30001"  ET 200SP-Station
   slot 0: "Rack_0"  Rack  6ES5 710-8MAx1
   slot 0: "n0048-lv002-el001-k30001"  IM 155-6 PN ST  6ES7 155-6AU01-0BN0  V4.2
   slot 1: "-K30002"  DI 16x24VDC ST  6ES7 131-6BH01-0BA0  V0.0
      slot 1: "-K30002"  DI 16x24VDC ST
   slot 2: "-K30003"  F-DI 8x24VDC HF  6ES7 136-6BA00-0CA0  V1.0
      slot 1: "-K30003"  F-DI 8x24VDC HF
   slot 3: "-K30004"  F-DQ 4x24VDC/2A PM HF  6ES7 136-6DB00-0CA0  V2.0
      slot 1: "-K30004"  F-DQ 4x24VDC/2A PM HF
   slot 4: "Server module_1"  Server module  6ES7 193-6PA00-0AA0  V1.1
      slot 1: "Server module_1"  Server module
   slot 127: "BA 2xRJ45"  BA 2xRJ45  6ES7 193-6AR00-0AA0  V0.0
      slot 1: "Port_1"  X1 P1 R  6ES7 193-6AR00-0AA0  V0.0
      slot 2: "Port_2"  X1 P2 R  6ES7 193-6AR00-0AA0  V0.0
DEVICE "n0050-uc13-el001-k30001"  ET 200SP-Station
   slot 0: "Rack_0"  Rack  6ES5 710-8MAx1
   slot 0: "n0050-uc13-el001-k30001"  IM 155-6 PN ST  6ES7 155-6AU01-0BN0  V4.2
   slot 1: "-K30002"  DI 16x24VDC ST  6ES7 131-6BH01-0BA0  V0.0
      slot 1: "-K30002"  DI 16x24VDC ST
   slot 2: "-K30003"  DI 16x24VDC ST  6ES7 131-6BH01-0BA0  V0.0
      slot 1: "-K30003"  DI 16x24VDC ST
   slot 3: "-K30004"  F-DI 8x24VDC HF  6ES7 136-6BA00-0CA0  V1.0
      slot 1: "-K30004"  F-DI 8x24VDC HF
   slot 4: "-K30005"  F-DI 8x24VDC HF  6ES7 136-6BA00-0CA0  V1.0
      slot 1: "-K30005"  F-DI 8x24VDC HF
   slot 5: "-K30006"  F-DI 8x24VDC HF  6ES7 136-6BA00-0CA0  V1.0
      slot 1: "-K30006"  F-DI 8x24VDC HF
   slot 6: "-K30007"  F-DI 8x24VDC HF  6ES7 136-6BA00-0CA0  V1.0
      slot 1: "-K30007"  F-DI 8x24VDC HF
   slot 7: "-K30008"  F-DQ 4x24VDC/2A PM HF  6ES7 136-6DB00-0CA0  V2.0
      slot 1: "-K30008"  F-DQ 4x24VDC/2A PM HF
   slot 8: "-K30009"  F-DQ 4x24VDC/2A PM HF  6ES7 136-6DB00-0CA0  V2.0
      slot 1: "-K30009"  F-DQ 4x24VDC/2A PM HF
   slot 9: "-K30010"  F-DQ 4x24VDC/2A PM HF  6ES7 136-6DB00-0CA0  V2.0
      slot 1: "-K30010"  F-DQ 4x24VDC/2A PM HF
   slot 10: "-K30011"  F-DQ 4x24VDC/2A PM HF  6ES7 136-6DB00-0CA0  V2.0
      slot 1: "-K30011"  F-DQ 4x24VDC/2A PM HF
   slot 11: "-K30012"  F-DQ 4x24VDC/2A PM HF  6ES7 136-6DB00-0CA0  V2.0
      slot 1: "-K30012"  F-DQ 4x24VDC/2A PM HF
   slot 12: "-K30013"  F-DQ 4x24VDC/2A PM HF  6ES7 136-6DB00-0CA0  V2.0
      slot 1: "-K30013"  F-DQ 4x24VDC/2A PM HF
   slot 13: "Server module_1"  Server module  6ES7 193-6PA00-0AA0  V1.1
      slot 1: "Server module_1"  Server module
   slot 127: "BA 2xRJ45"  BA 2xRJ45  6ES7 193-6AR00-0AA0  V0.0
      slot 1: "Port_1"  X1 P1 R  6ES7 193-6AR00-0AA0  V0.0
      slot 2: "Port_2"  X1 P2 R  6ES7 193-6AR00-0AA0  V0.0
DEVICE "n0051-uc134-xn10"  GSD.Device.PN
   slot 0: "Rack"  Rack  V1.0
   slot 0: "n0051-uc134-xn10"  55556 MVK-MPNIO F DI16/8  55556
      slot 0: "55556 MVK-MPNIO F DI16/8_1"  55556 MVK-MPNIO F DI16/8
      slot 1: "55556 MVK-MPNIO F DI16/8"  55556 MVK-MPNIO F DI16/8
         slot 1: "Port 1"  Port 1
         slot 2: "Port 2"  Port 2
      slot 1: "Power module_1"  Power module
         slot 0: "Power module"  Power module
   slot 2: "-XN10"  FS Data
      slot 0: "-XN10"  FS Data
DEVICE "n0053-uc12-el001-k30001"  ET 200SP-Station
   slot 0: "Rack_0"  Rack  6ES5 710-8MAx1
   slot 0: "n0053-uc12-el001-k30001"  IM 155-6 PN ST  6ES7 155-6AU01-0BN0  V4.2
   slot 1: "-K30002"  DI 16x24VDC ST  6ES7 131-6BH01-0BA0  V0.0
      slot 1: "-K30002"  DI 16x24VDC ST
   slot 2: "-K30003"  DI 16x24VDC ST  6ES7 131-6BH01-0BA0  V0.0
      slot 1: "-K30003"  DI 16x24VDC ST
   slot 3: "-K30004"  F-DI 8x24VDC HF  6ES7 136-6BA00-0CA0  V1.0
      slot 1: "-K30004"  F-DI 8x24VDC HF
   slot 4: "-K30005"  F-DI 8x24VDC HF  6ES7 136-6BA00-0CA0  V1.0
      slot 1: "-K30005"  F-DI 8x24VDC HF
   slot 5: "-K30006"  F-DI 8x24VDC HF  6ES7 136-6BA00-0CA0  V1.0
      slot 1: "-K30006"  F-DI 8x24VDC HF
   slot 6: "-K30007"  F-DI 8x24VDC HF  6ES7 136-6BA00-0CA0  V1.0
      slot 1: "-K30007"  F-DI 8x24VDC HF
   slot 7: "-K30008"  F-DQ 4x24VDC/2A PM HF  6ES7 136-6DB00-0CA0  V2.0
      slot 1: "-K30008"  F-DQ 4x24VDC/2A PM HF
   slot 8: "-K30009"  F-DQ 4x24VDC/2A PM HF  6ES7 136-6DB00-0CA0  V2.0
      slot 1: "-K30009"  F-DQ 4x24VDC/2A PM HF
   slot 9: "-K30010"  F-DQ 4x24VDC/2A PM HF  6ES7 136-6DB00-0CA0  V2.0
      slot 1: "-K30010"  F-DQ 4x24VDC/2A PM HF
   slot 10: "-K30011"  F-DQ 4x24VDC/2A PM HF  6ES7 136-6DB00-0CA0  V2.0
      slot 1: "-K30011"  F-DQ 4x24VDC/2A PM HF
   slot 11: "-K30012"  F-DQ 4x24VDC/2A PM HF  6ES7 136-6DB00-0CA0  V2.0
      slot 1: "-K30012"  F-DQ 4x24VDC/2A PM HF
   slot 12: "-K30013"  F-DQ 4x24VDC/2A PM HF  6ES7 136-6DB00-0CA0  V2.0
      slot 1: "-K30013"  F-DQ 4x24VDC/2A PM HF
   slot 13: "Server module_1"  Server module  6ES7 193-6PA00-0AA0  V1.1
      slot 1: "Server module_1"  Server module
   slot 127: "BA 2xRJ45"  BA 2xRJ45  6ES7 193-6AR00-0AA0  V0.0
      slot 1: "Port_1"  X1 P1 R  6ES7 193-6AR00-0AA0  V0.0
      slot 2: "Port_2"  X1 P2 R  6ES7 193-6AR00-0AA0  V0.0
DEVICE "n0055-uc124-xn10"  GSD.Device.PN
   slot 0: "Rack"  Rack  V1.0
   slot 0: "n0055-uc124-xn10"  55556 MVK-MPNIO F DI16/8  55556
      slot 0: "55556 MVK-MPNIO F DI16/8_1"  55556 MVK-MPNIO F DI16/8
      slot 1: "55556 MVK-MPNIO F DI16/8"  55556 MVK-MPNIO F DI16/8
         slot 1: "Port 1"  Port 1
         slot 2: "Port 2"  Port 2
      slot 1: "Power module_1"  Power module
         slot 0: "Power module"  Power module
   slot 2: "-XN10"  FS Data
      slot 0: "-XN10"  FS Data
DEVICE "n0054-uf31-el003-k30001"  ET 200SP-Station
   slot 0: "Rack_0"  Rack  6ES5 710-8MAx1
   slot 0: "n0054-uf31-el003-k30001"  IM 155-6 PN ST  6ES7 155-6AU01-0BN0  V4.2
   slot 1: "-K30002"  DI 16x24VDC ST  6ES7 131-6BH01-0BA0  V0.0
      slot 1: "-K30002"  DI 16x24VDC ST
   slot 2: "-K30003"  F-DI 8x24VDC HF  6ES7 136-6BA00-0CA0  V1.0
      slot 1: "-K30003"  F-DI 8x24VDC HF
   slot 3: "-K30004"  F-DQ 4x24VDC/2A PM HF  6ES7 136-6DB00-0CA0  V2.0
      slot 1: "-K30004"  F-DQ 4x24VDC/2A PM HF
   slot 4: "-K30005"  F-DQ 4x24VDC/2A PM HF  6ES7 136-6DB00-0CA0  V2.0
      slot 1: "-K30005"  F-DQ 4x24VDC/2A PM HF
   slot 5: "Server module_1"  Server module  6ES7 193-6PA00-0AA0  V1.1
      slot 1: "Server module_1"  Server module
   slot 127: "BA 2xRJ45"  BA 2xRJ45  6ES7 193-6AR00-0AA0  V0.0
      slot 1: "Port_1"  X1 P1 R  6ES7 193-6AR00-0AA0  V0.0
      slot 2: "Port_2"  X1 P2 R  6ES7 193-6AR00-0AA0  V0.0
DEVICE "n0057-uc11-el001-k30001"  ET 200SP-Station
   slot 0: "Rack_0"  Rack  6ES5 710-8MAx1
   slot 0: "n0057-uc11-el001-k30001"  IM 155-6 PN ST  6ES7 155-6AU01-0BN0  V4.2
   slot 1: "-K30002"  DI 16x24VDC ST  6ES7 131-6BH01-0BA0  V0.0
      slot 1: "-K30002"  DI 16x24VDC ST
   slot 2: "-K30003"  DI 16x24VDC ST  6ES7 131-6BH01-0BA0  V0.0
      slot 1: "-K30003"  DI 16x24VDC ST
   slot 3: "-K30004"  F-DI 8x24VDC HF  6ES7 136-6BA00-0CA0  V1.0
      slot 1: "-K30004"  F-DI 8x24VDC HF
   slot 4: "-K30005"  F-DI 8x24VDC HF  6ES7 136-6BA00-0CA0  V1.0
      slot 1: "-K30005"  F-DI 8x24VDC HF
   slot 5: "-K30006"  F-DI 8x24VDC HF  6ES7 136-6BA00-0CA0  V1.0
      slot 1: "-K30006"  F-DI 8x24VDC HF
   slot 6: "-K30007"  F-DI 8x24VDC HF  6ES7 136-6BA00-0CA0  V1.0
      slot 1: "-K30007"  F-DI 8x24VDC HF
   slot 7: "-K30008"  F-DQ 4x24VDC/2A PM HF  6ES7 136-6DB00-0CA0  V2.0
      slot 1: "-K30008"  F-DQ 4x24VDC/2A PM HF
   slot 8: "-K30009"  F-DQ 4x24VDC/2A PM HF  6ES7 136-6DB00-0CA0  V2.0
      slot 1: "-K30009"  F-DQ 4x24VDC/2A PM HF
   slot 9: "-K30010"  F-DQ 4x24VDC/2A PM HF  6ES7 136-6DB00-0CA0  V2.0
      slot 1: "-K30010"  F-DQ 4x24VDC/2A PM HF
   slot 10: "-K30011"  F-DQ 4x24VDC/2A PM HF  6ES7 136-6DB00-0CA0  V2.0
      slot 1: "-K30011"  F-DQ 4x24VDC/2A PM HF
   slot 11: "-K30012"  F-DQ 4x24VDC/2A PM HF  6ES7 136-6DB00-0CA0  V2.0
      slot 1: "-K30012"  F-DQ 4x24VDC/2A PM HF
   slot 12: "-K30013"  F-DQ 4x24VDC/2A PM HF  6ES7 136-6DB00-0CA0  V2.0
      slot 1: "-K30013"  F-DQ 4x24VDC/2A PM HF
   slot 13: "Server module_1"  Server module  6ES7 193-6PA00-0AA0  V1.1
      slot 1: "Server module_1"  Server module
   slot 127: "BA 2xRJ45"  BA 2xRJ45  6ES7 193-6AR00-0AA0  V0.0
      slot 1: "Port_1"  X1 P1 R  6ES7 193-6AR00-0AA0  V0.0
      slot 2: "Port_2"  X1 P2 R  6ES7 193-6AR00-0AA0  V0.0
DEVICE "n0060-uc114-xn10"  GSD.Device.PN
   slot 0: "Rack"  Rack  V1.0
   slot 0: "n0060-uc114-xn10"  55556 MVK-MPNIO F DI16/8  55556
      slot 0: "55556 MVK-MPNIO F DI16/8_1"  55556 MVK-MPNIO F DI16/8
      slot 1: "55556 MVK-MPNIO F DI16/8"  55556 MVK-MPNIO F DI16/8
         slot 1: "Port 1"  Port 1
         slot 2: "Port 2"  Port 2
      slot 1: "Power module_1"  Power module
         slot 0: "Power module"  Power module
   slot 2: "-XN10"  FS Data
      slot 0: "-XN10"  FS Data
DEVICE "n0058-lv003-el001-k30001"  ET 200SP-Station
   slot 0: "Rack_0"  Rack  6ES5 710-8MAx1
   slot 0: "n0058-lv003-el001-k30001"  IM 155-6 PN ST  6ES7 155-6AU01-0BN0  V4.2
   slot 1: "-K30002"  DI 16x24VDC ST  6ES7 131-6BH01-0BA0  V0.0
      slot 1: "-K30002"  DI 16x24VDC ST
   slot 2: "-K30003"  F-DI 8x24VDC HF  6ES7 136-6BA00-0CA0  V1.0
      slot 1: "-K30003"  F-DI 8x24VDC HF
   slot 3: "-K30004"  F-DQ 4x24VDC/2A PM HF  6ES7 136-6DB00-0CA0  V2.0
      slot 1: "-K30004"  F-DQ 4x24VDC/2A PM HF
   slot 4: "Server module_1"  Server module  6ES7 193-6PA00-0AA0  V1.1
      slot 1: "Server module_1"  Server module
   slot 127: "BA 2xRJ45"  BA 2xRJ45  6ES7 193-6AR00-0AA0  V0.0
      slot 1: "Port_1"  X1 P1 R  6ES7 193-6AR00-0AA0  V0.0
      slot 2: "Port_2"  X1 P2 R  6ES7 193-6AR00-0AA0  V0.0
DEVICE "n0059-lv003-el001-k30001"  ET 200SP-Station
   slot 0: "Rack_0"  Rack  6ES5 710-8MAx1
   slot 0: "n0059-lv003-el001-k30001"  IM 155-6 PN ST  6ES7 155-6AU01-0BN0  V4.2
   slot 1: "-K30002"  DI 16x24VDC ST  6ES7 131-6BH01-0BA0  V0.0
      slot 1: "-K30002"  DI 16x24VDC ST
   slot 2: "-K30003"  F-DI 8x24VDC HF  6ES7 136-6BA00-0CA0  V1.0
      slot 1: "-K30003"  F-DI 8x24VDC HF
   slot 3: "-K30004"  F-DQ 4x24VDC/2A PM HF  6ES7 136-6DB00-0CA0  V2.0
      slot 1: "-K30004"  F-DQ 4x24VDC/2A PM HF
   slot 4: "Server module_1"  Server module  6ES7 193-6PA00-0AA0  V1.1
      slot 1: "Server module_1"  Server module
   slot 127: "BA 2xRJ45"  BA 2xRJ45  6ES7 193-6AR00-0AA0  V0.0
      slot 1: "Port_1"  X1 P1 R  6ES7 193-6AR00-0AA0  V0.0
      slot 2: "Port_2"  X1 P2 R  6ES7 193-6AR00-0AA0  V0.0
DEVICE "n0028-uc17-el001-k30001"  ET 200SP-Station
   slot 0: "Rack_0"  Rack  6ES5 710-8MAx1
   slot 0: "n0028-uc17-el001-k30001"  IM 155-6 PN ST  6ES7 155-6AU01-0BN0  V4.2
   slot 1: "-K30002"  DI 16x24VDC ST  6ES7 131-6BH01-0BA0  V0.0
      slot 1: "-K30002"  DI 16x24VDC ST
   slot 2: "-K30003"  F-DI 8x24VDC HF  6ES7 136-6BA00-0CA0  V1.0
      slot 1: "-K30003"  F-DI 8x24VDC HF
   slot 3: "-K30004"  F-DI 8x24VDC HF  6ES7 136-6BA00-0CA0  V1.0
      slot 1: "-K30004"  F-DI 8x24VDC HF
   slot 4: "-K30005"  F-DI 8x24VDC HF  6ES7 136-6BA00-0CA0  V1.0
      slot 1: "-K30005"  F-DI 8x24VDC HF
   slot 5: "-K30006"  F-DQ 4x24VDC/2A PM HF  6ES7 136-6DB00-0CA0  V2.0
      slot 1: "-K30006"  F-DQ 4x24VDC/2A PM HF
   slot 6: "-K30007"  F-DQ 4x24VDC/2A PM HF  6ES7 136-6DB00-0CA0  V2.0
      slot 1: "-K30007"  F-DQ 4x24VDC/2A PM HF
   slot 7: "-K30008"  F-DQ 4x24VDC/2A PM HF  6ES7 136-6DB00-0CA0  V2.0
      slot 1: "-K30008"  F-DQ 4x24VDC/2A PM HF
   slot 8: "-K30009"  F-DQ 4x24VDC/2A PM HF  6ES7 136-6DB00-0CA0  V2.0
      slot 1: "-K30009"  F-DQ 4x24VDC/2A PM HF
   slot 9: "Server module_1"  Server module  6ES7 193-6PA00-0AA0  V1.1
      slot 1: "Server module_1"  Server module
   slot 127: "BA 2xRJ45"  BA 2xRJ45  6ES7 193-6AR00-0AA0  V0.0
      slot 1: "Port_1"  X1 P1 R  6ES7 193-6AR00-0AA0  V0.0
      slot 2: "Port_2"  X1 P2 R  6ES7 193-6AR00-0AA0  V0.0
DEVICE "n0029-uc173-xn10"  GSD.Device.PN
   slot 0: "Rack"  Rack  V1.0
   slot 0: "n0029-uc173-xn10"  55556 MVK-MPNIO F DI16/8  55556
      slot 0: "55556 MVK-MPNIO F DI16/8_1"  55556 MVK-MPNIO F DI16/8
      slot 1: "55556 MVK-MPNIO F DI16/8"  55556 MVK-MPNIO F DI16/8
         slot 1: "Port 1"  Port 1
         slot 2: "Port 2"  Port 2
      slot 1: "Power module_1"  Power module
         slot 0: "Power module"  Power module
   slot 2: "-XN10"  FS Data
      slot 0: "-XN10"  FS Data
DEVICE "n0010-zp001-el001-k24501"  PnPn.Device
   slot 0: "Rack"  Rail  1.0
   slot 0: "n0010-zp001-el001-k24501"  PN/PN Coupler  6ES7 158-3AD10-0XA0  V4.2
   slot 1: "UNDEFINED_3"  PN/PN Coupler  6ES7 158-3AD10-0XA0  V4.2
   slot 127: "BA 2xRJ45"  BA 2xRJ45  6ES7 193-6AR00-0AA0  V0.0
      slot 1: "Port_1"  X1 P1 R  6ES7 193-6AR00-0AA0  V0.0
      slot 2: "Port_2"  X1 P2 R  6ES7 193-6AR00-0AA0  V0.0
   slot 127: "BA 2xRJ45"  BA 2xRJ45  6ES7 193-6AR00-0AA0  V0.0
      slot 1: "Port_1"  X2 P1 R  6ES7 193-6AR00-0AA0  V0.0
      slot 2: "Port_2"  X2 P2 R  6ES7 193-6AR00-0AA0  V0.0
DEVICE "n0033-zp001-el001-k40001"  ET 200SP-Station
   slot 0: "Rack_0"  Rack  6ES5 710-8MAx1
   slot 0: "n0033-zp001-el001-k40001"  IM 155-6 PN ST  6ES7 155-6AU01-0BN0  V4.2
   slot 1: "-K40002"  DI 16x24VDC ST  6ES7 131-6BH01-0BA0  V0.0
      slot 1: "-K40002"  DI 16x24VDC ST
   slot 2: "-K40003"  F-DI 8x24VDC HF  6ES7 136-6BA00-0CA0  V1.0
      slot 1: "-K40003"  F-DI 8x24VDC HF
   slot 3: "-K40004"  F-DI 8x24VDC HF  6ES7 136-6BA00-0CA0  V1.0
      slot 1: "-K40004"  F-DI 8x24VDC HF
   slot 4: "-K40005"  F-DI 8x24VDC HF  6ES7 136-6BA00-0CA0  V1.0
      slot 1: "-K40005"  F-DI 8x24VDC HF
   slot 5: "-K40010"  F-DI 8x24VDC HF  6ES7 136-6BA00-0CA0  V1.0
      slot 1: "-K40010"  F-DI 8x24VDC HF
   slot 6: "-K40006"  F-DQ 4x24VDC/2A PM HF  6ES7 136-6DB00-0CA0  V2.0
      slot 1: "-K40006"  F-DQ 4x24VDC/2A PM HF
   slot 7: "-K40007"  F-DQ 4x24VDC/2A PM HF  6ES7 136-6DB00-0CA0  V2.0
      slot 1: "-K40007"  F-DQ 4x24VDC/2A PM HF
   slot 8: "-K40008"  F-DQ 4x24VDC/2A PM HF  6ES7 136-6DB00-0CA0  V2.0
      slot 1: "-K40008"  F-DQ 4x24VDC/2A PM HF
   slot 9: "-K40009"  DQ 16x24VDC/0.5A ST  6ES7 132-6BH01-0BA0  V0.0
      slot 1: "-K40009"  DQ 16x24VDC/0.5A ST
   slot 10: "Server module_1"  Server module  6ES7 193-6PA00-0AA0  V1.1
      slot 1: "Server module_1"  Server module
   slot 127: "BA 2xRJ45"  BA 2xRJ45  6ES7 193-6AR00-0AA0  V0.0
      slot 1: "Port_1"  X1 P1 R  6ES7 193-6AR00-0AA0  V0.0
      slot 2: "Port_2"  X1 P2 R  6ES7 193-6AR00-0AA0  V0.0
DEVICE "n0034-ug6-el001-k30001"  ET 200SP-Station
   slot 0: "Rack_0"  Rack  6ES5 710-8MAx1
   slot 0: "n0034-ug6-el001-k30001"  IM 155-6 PN ST  6ES7 155-6AU01-0BN0  V4.2
   slot 1: "-K30002"  DI 16x24VDC ST  6ES7 131-6BH01-0BA0  V0.0
      slot 1: "-K30002"  DI 16x24VDC ST
   slot 2: "-K30003"  DI 16x24VDC ST  6ES7 131-6BH01-0BA0  V0.0
      slot 1: "-K30003"  DI 16x24VDC ST
   slot 3: "-K30004"  F-DI 8x24VDC HF  6ES7 136-6BA00-0CA0  V1.0
      slot 1: "-K30004"  F-DI 8x24VDC HF
   slot 4: "-K30005"  F-DI 8x24VDC HF  6ES7 136-6BA00-0CA0  V1.0
      slot 1: "-K30005"  F-DI 8x24VDC HF
   slot 5: "-K30006"  F-DI 8x24VDC HF  6ES7 136-6BA00-0CA0  V1.0
      slot 1: "-K30006"  F-DI 8x24VDC HF
   slot 6: "-K30007"  F-DI 8x24VDC HF  6ES7 136-6BA00-0CA0  V1.0
      slot 1: "-K30007"  F-DI 8x24VDC HF
   slot 7: "-K30008"  F-DQ 4x24VDC/2A PM HF  6ES7 136-6DB00-0CA0  V2.0
      slot 1: "-K30008"  F-DQ 4x24VDC/2A PM HF
   slot 8: "-K30009"  F-DQ 4x24VDC/2A PM HF  6ES7 136-6DB00-0CA0  V2.0
      slot 1: "-K30009"  F-DQ 4x24VDC/2A PM HF
   slot 9: "-K30010"  F-DQ 4x24VDC/2A PM HF  6ES7 136-6DB00-0CA0  V2.0
      slot 1: "-K30010"  F-DQ 4x24VDC/2A PM HF
   slot 10: "-K30011"  F-DQ 4x24VDC/2A PM HF  6ES7 136-6DB00-0CA0  V2.0
      slot 1: "-K30011"  F-DQ 4x24VDC/2A PM HF
   slot 11: "-K30012"  F-DQ 4x24VDC/2A PM HF  6ES7 136-6DB00-0CA0  V2.0
      slot 1: "-K30012"  F-DQ 4x24VDC/2A PM HF
   slot 12: "-K30013"  F-DQ 4x24VDC/2A PM HF  6ES7 136-6DB00-0CA0  V2.0
      slot 1: "-K30013"  F-DQ 4x24VDC/2A PM HF
   slot 13: "-K30014"  F-DQ 4x24VDC/2A PM HF  6ES7 136-6DB00-0CA0  V2.0
      slot 1: "-K30014"  F-DQ 4x24VDC/2A PM HF
   slot 14: "Server module_1"  Server module  6ES7 193-6PA00-0AA0  V1.1
      slot 1: "Server module_1"  Server module
   slot 127: "BA 2xRJ45"  BA 2xRJ45  6ES7 193-6AR00-0AA0  V0.0
      slot 1: "Port_1"  X1 P1 R  6ES7 193-6AR00-0AA0  V0.0
      slot 2: "Port_2"  X1 P2 R  6ES7 193-6AR00-0AA0  V0.0
DEVICE "n0035-ug6-xn10"  GSD.Device.PN
   slot 0: "Rack"  Rack  V1.0
   slot 0: "n0035-ug6-xn10"  55556 MVK-MPNIO F DI16/8  55556
      slot 0: "55556 MVK-MPNIO F DI16/8_1"  55556 MVK-MPNIO F DI16/8
      slot 1: "55556 MVK-MPNIO F DI16/8"  55556 MVK-MPNIO F DI16/8
         slot 1: "Port 1"  Port 1
         slot 2: "Port 2"  Port 2
      slot 1: "Power module_1"  Power module
         slot 0: "Power module"  Power module
   slot 2: "-XN10"  FS Data
      slot 0: "-XN10"  FS Data
DEVICE "n0043-db93-el001-k30001"  ET 200SP-Station
   slot 0: "Rack_0"  Rack  6ES5 710-8MAx1
   slot 0: "n0043-db93-el001-k30001"  IM 155-6 PN ST  6ES7 155-6AU01-0BN0  V4.2
   slot 1: "-K30002"  DI 16x24VDC ST  6ES7 131-6BH01-0BA0  V0.0
      slot 1: "-K30002"  DI 16x24VDC ST
   slot 2: "-K30003"  F-DI 8x24VDC HF  6ES7 136-6BA00-0CA0  V1.0
      slot 1: "-K30003"  F-DI 8x24VDC HF
   slot 3: "-K30004"  F-DQ 4x24VDC/2A PM HF  6ES7 136-6DB00-0CA0  V2.0
      slot 1: "-K30004"  F-DQ 4x24VDC/2A PM HF
   slot 4: "Server module_1"  Server module  6ES7 193-6PA00-0AA0  V1.1
      slot 1: "Server module_1"  Server module
   slot 127: "BA 2xRJ45"  BA 2xRJ45  6ES7 193-6AR00-0AA0  V0.0
      slot 1: "Port_1"  X1 P1 R  6ES7 193-6AR00-0AA0  V0.0
      slot 2: "Port_2"  X1 P2 R  6ES7 193-6AR00-0AA0  V0.0
DEVICE "n0031-db931-xn10"  GSD.Device.PN
   slot 0: "Rack"  Rack  V1.0
   slot 0: "n0031-db931-xn10"  55556 MVK-MPNIO F DI16/8  55556
      slot 0: "55556 MVK-MPNIO F DI16/8_1"  55556 MVK-MPNIO F DI16/8
      slot 1: "55556 MVK-MPNIO F DI16/8"  55556 MVK-MPNIO F DI16/8
         slot 1: "Port 1"  Port 1
         slot 2: "Port 2"  Port 2
      slot 1: "Power module_1"  Power module
         slot 0: "Power module"  Power module
   slot 2: "-XN10"  FS Data
      slot 0: "-XN10"  FS Data
DEVICE "n0005-lv008-el001-k30001"  ET 200SP-Station
   slot 0: "Rack_0"  Rack  6ES5 710-8MAx1
   slot 0: "n0005-lv008-el001-k30001"  IM 155-6 PN ST  6ES7 155-6AU01-0BN0  V4.2
   slot 1: "-K30002"  DI 16x24VDC ST  6ES7 131-6BH01-0BA0  V0.0
      slot 1: "-K30002"  DI 16x24VDC ST
   slot 2: "-K30003"  F-DI 8x24VDC HF  6ES7 136-6BA00-0CA0  V1.0
      slot 1: "-K30003"  F-DI 8x24VDC HF
   slot 3: "-K30004"  F-DI 8x24VDC HF  6ES7 136-6BA00-0CA0  V1.0
      slot 1: "-K30004"  F-DI 8x24VDC HF
   slot 4: "-K30005"  F-DQ 4x24VDC/2A PM HF  6ES7 136-6DB00-0CA0  V2.0
      slot 1: "-K30005"  F-DQ 4x24VDC/2A PM HF
   slot 5: "-K30006"  F-DQ 4x24VDC/2A PM HF  6ES7 136-6DB00-0CA0  V2.0
      slot 1: "-K30006"  F-DQ 4x24VDC/2A PM HF
   slot 6: "Server module_1"  Server module  6ES7 193-6PA00-0AA0  V1.1
      slot 1: "Server module_1"  Server module
   slot 127: "BA 2xRJ45"  BA 2xRJ45  6ES7 193-6AR00-0AA0  V0.0
      slot 1: "Port_1"  X1 P1 R  6ES7 193-6AR00-0AA0  V0.0
      slot 2: "Port_2"  X1 P2 R  6ES7 193-6AR00-0AA0  V0.0
DEVICE "n0006-lv008-el001-k30001"  ET 200SP-Station
   slot 0: "Rack_0"  Rack  6ES5 710-8MAx1
   slot 0: "n0006-lv008-el001-k30001"  IM 155-6 PN ST  6ES7 155-6AU01-0BN0  V4.2
   slot 1: "-K30002"  DI 16x24VDC ST  6ES7 131-6BH01-0BA0  V0.0
      slot 1: "-K30002"  DI 16x24VDC ST
   slot 2: "-K30003"  F-DI 8x24VDC HF  6ES7 136-6BA00-0CA0  V1.0
      slot 1: "-K30003"  F-DI 8x24VDC HF
   slot 3: "-K30004"  F-DI 8x24VDC HF  6ES7 136-6BA00-0CA0  V1.0
      slot 1: "-K30004"  F-DI 8x24VDC HF
   slot 4: "-K30005"  F-DQ 4x24VDC/2A PM HF  6ES7 136-6DB00-0CA0  V2.0
      slot 1: "-K30005"  F-DQ 4x24VDC/2A PM HF
   slot 5: "-K30006"  F-DQ 4x24VDC/2A PM HF  6ES7 136-6DB00-0CA0  V2.0
      slot 1: "-K30006"  F-DQ 4x24VDC/2A PM HF
   slot 6: "Server module_1"  Server module  6ES7 193-6PA00-0AA0  V1.1
      slot 1: "Server module_1"  Server module
   slot 127: "BA 2xRJ45"  BA 2xRJ45  6ES7 193-6AR00-0AA0  V0.0
      slot 1: "Port_1"  X1 P1 R  6ES7 193-6AR00-0AA0  V0.0
      slot 2: "Port_2"  X1 P2 R  6ES7 193-6AR00-0AA0  V0.0
DEVICE "n0007-icg22-el001-k30001"  ET 200SP-Station
   slot 0: "Rack_0"  Rack  6ES5 710-8MAx1
   slot 0: "n0007-icg22-el001-k30001"  IM 155-6 PN ST  6ES7 155-6AU01-0BN0  V4.2
   slot 1: "-K30002"  DI 16x24VDC ST  6ES7 131-6BH01-0BA0  V0.0
      slot 1: "-K30002"  DI 16x24VDC ST
   slot 2: "-K30003"  F-DI 8x24VDC HF  6ES7 136-6BA00-0CA0  V1.0
      slot 1: "-K30003"  F-DI 8x24VDC HF
   slot 3: "-K30004"  F-DI 8x24VDC HF  6ES7 136-6BA00-0CA0  V1.0
      slot 1: "-K30004"  F-DI 8x24VDC HF
   slot 4: "-K30005"  F-DI 8x24VDC HF  6ES7 136-6BA00-0CA0  V1.0
      slot 1: "-K30005"  F-DI 8x24VDC HF
   slot 5: "-K30006"  F-DI 8x24VDC HF  6ES7 136-6BA00-0CA0  V1.0
      slot 1: "-K30006"  F-DI 8x24VDC HF
   slot 6: "-K30007"  F-DQ 4x24VDC/2A PM HF  6ES7 136-6DB00-0CA0  V2.0
      slot 1: "-K30007"  F-DQ 4x24VDC/2A PM HF
   slot 7: "-K30008"  F-DQ 4x24VDC/2A PM HF  6ES7 136-6DB00-0CA0  V2.0
      slot 1: "-K30008"  F-DQ 4x24VDC/2A PM HF
   slot 8: "-K30009"  F-DQ 4x24VDC/2A PM HF  6ES7 136-6DB00-0CA0  V2.0
      slot 1: "-K30009"  F-DQ 4x24VDC/2A PM HF
   slot 9: "Server module_1"  Server module  6ES7 193-6PA00-0AA0  V1.1
      slot 1: "Server module_1"  Server module
   slot 127: "BA 2xRJ45"  BA 2xRJ45  6ES7 193-6AR00-0AA0  V0.0
      slot 1: "Port_1"  X1 P1 R  6ES7 193-6AR00-0AA0  V0.0
      slot 2: "Port_2"  X1 P2 R  6ES7 193-6AR00-0AA0  V0.0
DEVICE "n0008-icg12-el001-k30001"  ET 200SP-Station
   slot 0: "Rack_0"  Rack  6ES5 710-8MAx1
   slot 0: "n0008-icg12-el001-k30001"  IM 155-6 PN ST  6ES7 155-6AU01-0BN0  V4.2
   slot 1: "-K30002"  DI 16x24VDC ST  6ES7 131-6BH01-0BA0  V0.0
      slot 1: "-K30002"  DI 16x24VDC ST
   slot 2: "-K30003"  F-DI 8x24VDC HF  6ES7 136-6BA00-0CA0  V1.0
      slot 1: "-K30003"  F-DI 8x24VDC HF
   slot 3: "-K30004"  F-DI 8x24VDC HF  6ES7 136-6BA00-0CA0  V1.0
      slot 1: "-K30004"  F-DI 8x24VDC HF
   slot 4: "-K30005"  F-DI 8x24VDC HF  6ES7 136-6BA00-0CA0  V1.0
      slot 1: "-K30005"  F-DI 8x24VDC HF
   slot 5: "-K30006"  F-DI 8x24VDC HF  6ES7 136-6BA00-0CA0  V1.0
      slot 1: "-K30006"  F-DI 8x24VDC HF
   slot 6: "-K30007"  F-DQ 4x24VDC/2A PM HF  6ES7 136-6DB00-0CA0  V2.0
      slot 1: "-K30007"  F-DQ 4x24VDC/2A PM HF
   slot 7: "-K30008"  F-DQ 4x24VDC/2A PM HF  6ES7 136-6DB00-0CA0  V2.0
      slot 1: "-K30008"  F-DQ 4x24VDC/2A PM HF
   slot 8: "-K30009"  F-DQ 4x24VDC/2A PM HF  6ES7 136-6DB00-0CA0  V2.0
      slot 1: "-K30009"  F-DQ 4x24VDC/2A PM HF
   slot 9: "Server module_1"  Server module  6ES7 193-6PA00-0AA0  V1.1
      slot 1: "Server module_1"  Server module
   slot 127: "BA 2xRJ45"  BA 2xRJ45  6ES7 193-6AR00-0AA0  V0.0
      slot 1: "Port_1"  X1 P1 R  6ES7 193-6AR00-0AA0  V0.0
      slot 2: "Port_2"  X1 P2 R  6ES7 193-6AR00-0AA0  V0.0
DEVICE "n0009-uf42-el002-k30001"  ET 200SP-Station
   slot 0: "Rack_0"  Rack  6ES5 710-8MAx1
   slot 0: "n0009-uf42-el002-k30001"  IM 155-6 PN ST  6ES7 155-6AU01-0BN0  V4.2
   slot 1: "-K30002"  DI 16x24VDC ST  6ES7 131-6BH01-0BA0  V0.0
      slot 1: "-K30002"  DI 16x24VDC ST
   slot 2: "-K30003"  F-DI 8x24VDC HF  6ES7 136-6BA00-0CA0  V1.0
      slot 1: "-K30003"  F-DI 8x24VDC HF
   slot 3: "-K30004"  F-DQ 4x24VDC/2A PM HF  6ES7 136-6DB00-0CA0  V2.0
      slot 1: "-K30004"  F-DQ 4x24VDC/2A PM HF
   slot 4: "-K30005"  F-DQ 4x24VDC/2A PM HF  6ES7 136-6DB00-0CA0  V2.0
      slot 1: "-K30005"  F-DQ 4x24VDC/2A PM HF
   slot 5: "Server module_1"  Server module  6ES7 193-6PA00-0AA0  V1.1
      slot 1: "Server module_1"  Server module
   slot 127: "BA 2xRJ45"  BA 2xRJ45  6ES7 193-6AR00-0AA0  V0.0
      slot 1: "Port_1"  X1 P1 R  6ES7 193-6AR00-0AA0  V0.0
      slot 2: "Port_2"  X1 P2 R  6ES7 193-6AR00-0AA0  V0.0
DEVICE "n0010-lv007-el001-k30001"  ET 200SP-Station
   slot 0: "Rack_0"  Rack  6ES5 710-8MAx1
   slot 0: "n0010-lv007-el001-k30001"  IM 155-6 PN ST  6ES7 155-6AU01-0BN0  V4.2
   slot 1: "-K30002"  DI 16x24VDC ST  6ES7 131-6BH01-0BA0  V0.0
      slot 1: "-K30002"  DI 16x24VDC ST
   slot 2: "-K30003"  F-DI 8x24VDC HF  6ES7 136-6BA00-0CA0  V1.0
      slot 1: "-K30003"  F-DI 8x24VDC HF
   slot 3: "-K30004"  F-DQ 4x24VDC/2A PM HF  6ES7 136-6DB00-0CA0  V2.0
      slot 1: "-K30004"  F-DQ 4x24VDC/2A PM HF
   slot 4: "Server module_1"  Server module  6ES7 193-6PA00-0AA0  V1.1
      slot 1: "Server module_1"  Server module
   slot 127: "BA 2xRJ45"  BA 2xRJ45  6ES7 193-6AR00-0AA0  V0.0
      slot 1: "Port_1"  X1 P1 R  6ES7 193-6AR00-0AA0  V0.0
      slot 2: "Port_2"  X1 P2 R  6ES7 193-6AR00-0AA0  V0.0
DEVICE "n0011-lv007-el001-k30001"  ET 200SP-Station
   slot 0: "Rack_0"  Rack  6ES5 710-8MAx1
   slot 0: "n0011-lv007-el001-k30001"  IM 155-6 PN ST  6ES7 155-6AU01-0BN0  V4.2
   slot 1: "-K30002"  DI 16x24VDC ST  6ES7 131-6BH01-0BA0  V0.0
      slot 1: "-K30002"  DI 16x24VDC ST
   slot 2: "-K30003"  F-DI 8x24VDC HF  6ES7 136-6BA00-0CA0  V1.0
      slot 1: "-K30003"  F-DI 8x24VDC HF
   slot 3: "-K30004"  F-DQ 4x24VDC/2A PM HF  6ES7 136-6DB00-0CA0  V2.0
      slot 1: "-K30004"  F-DQ 4x24VDC/2A PM HF
   slot 4: "Server module_1"  Server module  6ES7 193-6PA00-0AA0  V1.1
      slot 1: "Server module_1"  Server module
   slot 127: "BA 2xRJ45"  BA 2xRJ45  6ES7 193-6AR00-0AA0  V0.0
      slot 1: "Port_1"  X1 P1 R  6ES7 193-6AR00-0AA0  V0.0
      slot 2: "Port_2"  X1 P2 R  6ES7 193-6AR00-0AA0  V0.0
DEVICE "n0021-uc2-el001-k30001"  ET 200SP-Station
   slot 0: "Rack_0"  Rack  6ES5 710-8MAx1
   slot 0: "n0021-uc2-el001-k30001"  IM 155-6 PN ST  6ES7 155-6AU01-0BN0  V4.2
   slot 1: "-K30002"  DI 16x24VDC ST  6ES7 131-6BH01-0BA0  V0.0
      slot 1: "-K30002"  DI 16x24VDC ST
   slot 2: "-K30003"  F-DI 8x24VDC HF  6ES7 136-6BA00-0CA0  V1.0
      slot 1: "-K30003"  F-DI 8x24VDC HF
   slot 3: "-K30004"  F-DQ 4x24VDC/2A PM HF  6ES7 136-6DB00-0CA0  V2.0
      slot 1: "-K30004"  F-DQ 4x24VDC/2A PM HF
   slot 4: "-K30005"  DQ 16x24VDC/0.5A ST  6ES7 132-6BH01-0BA0  V0.0
      slot 1: "-K30005"  DQ 16x24VDC/0.5A ST
   slot 5: "Server module_1"  Server module  6ES7 193-6PA00-0AA0  V1.1
      slot 1: "Server module_1"  Server module
   slot 127: "BA 2xRJ45"  BA 2xRJ45  6ES7 193-6AR00-0AA0  V0.0
      slot 1: "Port_1"  X1 P1 R  6ES7 193-6AR00-0AA0  V0.0
      slot 2: "Port_2"  X1 P2 R  6ES7 193-6AR00-0AA0  V0.0
DEVICE "n0025-dc91-el001-k30001"  ET 200SP-Station
   slot 0: "Rack_0"  Rack  6ES5 710-8MAx1
   slot 0: "n0025-dc91-el001-k30001"  IM 155-6 PN ST  6ES7 155-6AU01-0BN0  V4.2
   slot 1: "-K30002"  DI 16x24VDC ST  6ES7 131-6BH01-0BA0  V0.0
      slot 1: "-K30002"  DI 16x24VDC ST
   slot 2: "-K30003"  F-DI 8x24VDC HF  6ES7 136-6BA00-0CA0  V1.0
      slot 1: "-K30003"  F-DI 8x24VDC HF
   slot 3: "-K30004"  F-DQ 4x24VDC/2A PM HF  6ES7 136-6DB00-0CA0  V2.0
      slot 1: "-K30004"  F-DQ 4x24VDC/2A PM HF
   slot 4: "-K30005"  F-DQ 4x24VDC/2A PM HF  6ES7 136-6DB00-0CA0  V2.0
      slot 1: "-K30005"  F-DQ 4x24VDC/2A PM HF
   slot 5: "-K30006"  F-DQ 4x24VDC/2A PM HF  6ES7 136-6DB00-0CA0  V2.0
      slot 1: "-K30006"  F-DQ 4x24VDC/2A PM HF
   slot 6: "Server module_1"  Server module  6ES7 193-6PA00-0AA0  V1.1
      slot 1: "Server module_1"  Server module
   slot 127: "BA 2xRJ45"  BA 2xRJ45  6ES7 193-6AR00-0AA0  V0.0
      slot 1: "Port_1"  X1 P1 R  6ES7 193-6AR00-0AA0  V0.0
      slot 2: "Port_2"  X1 P2 R  6ES7 193-6AR00-0AA0  V0.0
DEVICE "n0026-uc915-xn10"  GSD.Device.PN
   slot 0: "Rack"  Rack  V1.0
   slot 0: "n0026-uc915-xn10"  55556 MVK-MPNIO F DI16/8  55556
      slot 0: "55556 MVK-MPNIO F DI16/8_1"  55556 MVK-MPNIO F DI16/8
      slot 1: "55556 MVK-MPNIO F DI16/8"  55556 MVK-MPNIO F DI16/8
         slot 1: "Port 1"  Port 1
         slot 2: "Port 2"  Port 2
      slot 1: "Power module_1"  Power module
         slot 0: "Power module"  Power module
   slot 2: "-XN10"  FS Data
      slot 0: "-XN10"  FS Data
DEVICE "n0027-uc915-xn11"  GSD.Device.PN
   slot 0: "Rack"  Rack  V1.0
   slot 0: "n0027-uc915-xn11"  55556 MVK-MPNIO F DI16/8  55556
      slot 0: "55556 MVK-MPNIO F DI16/8_1"  55556 MVK-MPNIO F DI16/8
      slot 1: "55556 MVK-MPNIO F DI16/8"  55556 MVK-MPNIO F DI16/8
         slot 1: "Port 1"  Port 1
         slot 2: "Port 2"  Port 2
      slot 1: "Power module_1"  Power module
         slot 0: "Power module"  Power module
   slot 2: "-XN11"  FS Data
      slot 0: "-XN11"  FS Data
DEVICE "n0028-lv005-el001-k30001"  ET 200SP-Station
   slot 0: "Rack_0"  Rack  6ES5 710-8MAx1
   slot 0: "n0028-lv005-el001-k30001"  IM 155-6 PN ST  6ES7 155-6AU01-0BN0  V4.2
   slot 1: "-K30002"  DI 16x24VDC ST  6ES7 131-6BH01-0BA0  V0.0
      slot 1: "-K30002"  DI 16x24VDC ST
   slot 2: "-K30003"  F-DI 8x24VDC HF  6ES7 136-6BA00-0CA0  V1.0
      slot 1: "-K30003"  F-DI 8x24VDC HF
   slot 3: "-K30004"  F-DQ 4x24VDC/2A PM HF  6ES7 136-6DB00-0CA0  V2.0
      slot 1: "-K30004"  F-DQ 4x24VDC/2A PM HF
   slot 4: "Server module_1"  Server module  6ES7 193-6PA00-0AA0  V1.1
      slot 1: "Server module_1"  Server module
   slot 127: "BA 2xRJ45"  BA 2xRJ45  6ES7 193-6AR00-0AA0  V0.0
      slot 1: "Port_1"  X1 P1 R  6ES7 193-6AR00-0AA0  V0.0
      slot 2: "Port_2"  X1 P2 R  6ES7 193-6AR00-0AA0  V0.0
DEVICE "n0029-ct2-el001-k30001"  ET 200SP-Station
   slot 0: "Rack_0"  Rack  6ES5 710-8MAx1
   slot 0: "n0029-ct2-el001-k30001"  IM 155-6 PN ST  6ES7 155-6AU01-0BN0  V4.2
   slot 1: "-K30002"  DI 16x24VDC ST  6ES7 131-6BH01-0BA0  V0.0
      slot 1: "-K30002"  DI 16x24VDC ST
   slot 2: "-K30003"  F-DI 8x24VDC HF  6ES7 136-6BA00-0CA0  V1.0
      slot 1: "-K30003"  F-DI 8x24VDC HF
   slot 3: "-K30004"  F-DI 8x24VDC HF  6ES7 136-6BA00-0CA0  V1.0
      slot 1: "-K30004"  F-DI 8x24VDC HF
   slot 4: "-K30005"  F-DI 8x24VDC HF  6ES7 136-6BA00-0CA0  V1.0
      slot 1: "-K30005"  F-DI 8x24VDC HF
   slot 5: "-K30006"  F-DI 8x24VDC HF  6ES7 136-6BA00-0CA0  V1.0
      slot 1: "-K30006"  F-DI 8x24VDC HF
   slot 6: "-K30007"  F-DI 8x24VDC HF  6ES7 136-6BA00-0CA0  V1.0
      slot 1: "-K30007"  F-DI 8x24VDC HF
   slot 7: "-K30008"  F-DQ 4x24VDC/2A PM HF  6ES7 136-6DB00-0CA0  V2.0
      slot 1: "-K30008"  F-DQ 4x24VDC/2A PM HF
   slot 8: "-K30009"  F-DQ 4x24VDC/2A PM HF  6ES7 136-6DB00-0CA0  V2.0
      slot 1: "-K30009"  F-DQ 4x24VDC/2A PM HF
   slot 9: "Server module_1"  Server module  6ES7 193-6PA00-0AA0  V1.1
      slot 1: "Server module_1"  Server module
   slot 127: "BA 2xRJ45"  BA 2xRJ45  6ES7 193-6AR00-0AA0  V0.0
      slot 1: "Port_1"  X1 P1 R  6ES7 193-6AR00-0AA0  V0.0
      slot 2: "Port_2"  X1 P2 R  6ES7 193-6AR00-0AA0  V0.0
DEVICE "n0033-uc26-el001-k30001"  ET 200SP-Station
   slot 0: "Rack_0"  Rack  6ES5 710-8MAx1
   slot 0: "n0033-uc26-el001-k30001"  IM 155-6 PN ST  6ES7 155-6AU01-0BN0  V4.2
   slot 1: "-K30002"  DI 16x24VDC ST  6ES7 131-6BH01-0BA0  V0.0
      slot 1: "-K30002"  DI 16x24VDC ST
   slot 2: "-K30003"  DI 16x24VDC ST  6ES7 131-6BH01-0BA0  V0.0
      slot 1: "-K30003"  DI 16x24VDC ST
   slot 3: "-K30004"  F-DI 8x24VDC HF  6ES7 136-6BA00-0CA0  V1.0
      slot 1: "-K30004"  F-DI 8x24VDC HF
   slot 4: "-K30005"  F-DI 8x24VDC HF  6ES7 136-6BA00-0CA0  V1.0
      slot 1: "-K30005"  F-DI 8x24VDC HF
   slot 5: "-K30006"  F-DI 8x24VDC HF  6ES7 136-6BA00-0CA0  V1.0
      slot 1: "-K30006"  F-DI 8x24VDC HF
   slot 6: "-K30007"  F-DI 8x24VDC HF  6ES7 136-6BA00-0CA0  V1.0
      slot 1: "-K30007"  F-DI 8x24VDC HF
   slot 7: "-K30008"  F-DQ 4x24VDC/2A PM HF  6ES7 136-6DB00-0CA0  V2.0
      slot 1: "-K30008"  F-DQ 4x24VDC/2A PM HF
   slot 8: "-K30009"  F-DQ 4x24VDC/2A PM HF  6ES7 136-6DB00-0CA0  V2.0
      slot 1: "-K30009"  F-DQ 4x24VDC/2A PM HF
   slot 9: "-K30010"  F-DQ 4x24VDC/2A PM HF  6ES7 136-6DB00-0CA0  V2.0
      slot 1: "-K30010"  F-DQ 4x24VDC/2A PM HF
   slot 10: "-K30011"  F-DQ 4x24VDC/2A PM HF  6ES7 136-6DB00-0CA0  V2.0
      slot 1: "-K30011"  F-DQ 4x24VDC/2A PM HF
   slot 11: "-K30012"  F-DQ 4x24VDC/2A PM HF  6ES7 136-6DB00-0CA0  V2.0
      slot 1: "-K30012"  F-DQ 4x24VDC/2A PM HF
   slot 12: "-K30013"  F-DQ 4x24VDC/2A PM HF  6ES7 136-6DB00-0CA0  V2.0
      slot 1: "-K30013"  F-DQ 4x24VDC/2A PM HF
   slot 13: "Server module_1"  Server module  6ES7 193-6PA00-0AA0  V1.1
      slot 1: "Server module_1"  Server module
   slot 127: "BA 2xRJ45"  BA 2xRJ45  6ES7 193-6AR00-0AA0  V0.0
      slot 1: "Port_1"  X1 P1 R  6ES7 193-6AR00-0AA0  V0.0
      slot 2: "Port_2"  X1 P2 R  6ES7 193-6AR00-0AA0  V0.0
DEVICE "n0034-uc264-xn10"  GSD.Device.PN
   slot 0: "Rack"  Rack  V1.0
   slot 0: "n0034-uc264-xn10"  55556 MVK-MPNIO F DI16/8  55556
      slot 0: "55556 MVK-MPNIO F DI16/8_1"  55556 MVK-MPNIO F DI16/8
      slot 1: "55556 MVK-MPNIO F DI16/8"  55556 MVK-MPNIO F DI16/8
         slot 1: "Port 1"  Port 1
         slot 2: "Port 2"  Port 2
      slot 1: "Power module_1"  Power module
         slot 0: "Power module"  Power module
   slot 2: "-XN10"  FS Data
      slot 0: "-XN10"  FS Data
DEVICE "n0035-ct2-el002-k30001"  ET 200SP-Station
   slot 0: "Rack_0"  Rack  6ES5 710-8MAx1
   slot 0: "n0035-ct2-el002-k30001"  IM 155-6 PN ST  6ES7 155-6AU01-0BN0  V4.2
   slot 1: "-K30002"  DI 16x24VDC ST  6ES7 131-6BH01-0BA0  V0.0
      slot 1: "-K30002"  DI 16x24VDC ST
   slot 2: "-K30003"  F-DI 8x24VDC HF  6ES7 136-6BA00-0CA0  V1.0
      slot 1: "-K30003"  F-DI 8x24VDC HF
   slot 3: "-K30004"  F-DI 8x24VDC HF  6ES7 136-6BA00-0CA0  V1.0
      slot 1: "-K30004"  F-DI 8x24VDC HF
   slot 4: "-K30005"  F-DI 8x24VDC HF  6ES7 136-6BA00-0CA0  V1.0
      slot 1: "-K30005"  F-DI 8x24VDC HF
   slot 5: "-K30006"  F-DI 8x24VDC HF  6ES7 136-6BA00-0CA0  V1.0
      slot 1: "-K30006"  F-DI 8x24VDC HF
   slot 6: "-K30007"  F-DI 8x24VDC HF  6ES7 136-6BA00-0CA0  V1.0
      slot 1: "-K30007"  F-DI 8x24VDC HF
   slot 7: "-K30008"  F-DQ 4x24VDC/2A PM HF  6ES7 136-6DB00-0CA0  V2.0
      slot 1: "-K30008"  F-DQ 4x24VDC/2A PM HF
   slot 8: "-K30009"  F-DQ 4x24VDC/2A PM HF  6ES7 136-6DB00-0CA0  V2.0
      slot 1: "-K30009"  F-DQ 4x24VDC/2A PM HF
   slot 9: "Server module_1"  Server module  6ES7 193-6PA00-0AA0  V1.1
      slot 1: "Server module_1"  Server module
   slot 127: "BA 2xRJ45"  BA 2xRJ45  6ES7 193-6AR00-0AA0  V0.0
      slot 1: "Port_1"  X1 P1 R  6ES7 193-6AR00-0AA0  V0.0
      slot 2: "Port_2"  X1 P2 R  6ES7 193-6AR00-0AA0  V0.0
DEVICE "n0036-lv005-el001-k30001"  ET 200SP-Station
   slot 0: "Rack_0"  Rack  6ES5 710-8MAx1
   slot 0: "n0036-lv005-el001-k30001"  IM 155-6 PN ST  6ES7 155-6AU01-0BN0  V4.2
   slot 1: "-K30002"  DI 16x24VDC ST  6ES7 131-6BH01-0BA0  V0.0
      slot 1: "-K30002"  DI 16x24VDC ST
   slot 2: "-K30003"  F-DI 8x24VDC HF  6ES7 136-6BA00-0CA0  V1.0
      slot 1: "-K30003"  F-DI 8x24VDC HF
   slot 3: "-K30004"  F-DQ 4x24VDC/2A PM HF  6ES7 136-6DB00-0CA0  V2.0
      slot 1: "-K30004"  F-DQ 4x24VDC/2A PM HF
   slot 4: "Server module_1"  Server module  6ES7 193-6PA00-0AA0  V1.1
      slot 1: "Server module_1"  Server module
   slot 127: "BA 2xRJ45"  BA 2xRJ45  6ES7 193-6AR00-0AA0  V0.0
      slot 1: "Port_1"  X1 P1 R  6ES7 193-6AR00-0AA0  V0.0
      slot 2: "Port_2"  X1 P2 R  6ES7 193-6AR00-0AA0  V0.0
DEVICE "n0041-uc27-el001-k30001"  ET 200SP-Station
   slot 0: "Rack_0"  Rack  6ES5 710-8MAx1
   slot 0: "n0041-uc27-el001-k30001"  IM 155-6 PN ST  6ES7 155-6AU01-0BN0  V4.2
   slot 1: "-K30002"  DI 16x24VDC ST  6ES7 131-6BH01-0BA0  V0.0
      slot 1: "-K30002"  DI 16x24VDC ST
   slot 2: "-K30003"  F-DI 8x24VDC HF  6ES7 136-6BA00-0CA0  V1.0
      slot 1: "-K30003"  F-DI 8x24VDC HF
   slot 3: "-K30004"  F-DI 8x24VDC HF  6ES7 136-6BA00-0CA0  V1.0
      slot 1: "-K30004"  F-DI 8x24VDC HF
   slot 4: "-K30005"  F-DI 8x24VDC HF  6ES7 136-6BA00-0CA0  V1.0
      slot 1: "-K30005"  F-DI 8x24VDC HF
   slot 5: "-K30006"  F-DQ 4x24VDC/2A PM HF  6ES7 136-6DB00-0CA0  V2.0
      slot 1: "-K30006"  F-DQ 4x24VDC/2A PM HF
   slot 6: "-K30007"  F-DQ 4x24VDC/2A PM HF  6ES7 136-6DB00-0CA0  V2.0
      slot 1: "-K30007"  F-DQ 4x24VDC/2A PM HF
   slot 7: "-K30008"  F-DQ 4x24VDC/2A PM HF  6ES7 136-6DB00-0CA0  V2.0
      slot 1: "-K30008"  F-DQ 4x24VDC/2A PM HF
   slot 8: "-K30009"  F-DQ 4x24VDC/2A PM HF  6ES7 136-6DB00-0CA0  V2.0
      slot 1: "-K30009"  F-DQ 4x24VDC/2A PM HF
   slot 9: "Server module_1"  Server module  6ES7 193-6PA00-0AA0  V1.1
      slot 1: "Server module_1"  Server module
   slot 127: "BA 2xRJ45"  BA 2xRJ45  6ES7 193-6AR00-0AA0  V0.0
      slot 1: "Port_1"  X1 P1 R  6ES7 193-6AR00-0AA0  V0.0
      slot 2: "Port_2"  X1 P2 R  6ES7 193-6AR00-0AA0  V0.0
DEVICE "n0042-uc274-xn10"  GSD.Device.PN
   slot 0: "Rack"  Rack  V1.0
   slot 0: "n0042-uc274-xn10"  55556 MVK-MPNIO F DI16/8  55556
      slot 0: "55556 MVK-MPNIO F DI16/8_1"  55556 MVK-MPNIO F DI16/8
      slot 1: "55556 MVK-MPNIO F DI16/8"  55556 MVK-MPNIO F DI16/8
         slot 1: "Port 1"  Port 1
         slot 2: "Port 2"  Port 2
      slot 1: "Power module_1"  Power module
         slot 0: "Power module"  Power module
   slot 2: "-XN10"  FS Data
      slot 0: "-XN10"  FS Data
DEVICE "n0046-uc25-el001-k30001"  ET 200SP-Station
   slot 0: "Rack_0"  Rack  6ES5 710-8MAx1
   slot 0: "n0046-uc25-el001-k30001"  IM 155-6 PN ST  6ES7 155-6AU01-0BN0  V4.2
   slot 1: "-K30002"  DI 16x24VDC ST  6ES7 131-6BH01-0BA0  V0.0
      slot 1: "-K30002"  DI 16x24VDC ST
   slot 2: "-K30003"  DI 16x24VDC ST  6ES7 131-6BH01-0BA0  V0.0
      slot 1: "-K30003"  DI 16x24VDC ST
   slot 3: "-K30004"  F-DI 8x24VDC HF  6ES7 136-6BA00-0CA0  V1.0
      slot 1: "-K30004"  F-DI 8x24VDC HF
   slot 4: "-K30005"  F-DI 8x24VDC HF  6ES7 136-6BA00-0CA0  V1.0
      slot 1: "-K30005"  F-DI 8x24VDC HF
   slot 5: "-K30006"  F-DI 8x24VDC HF  6ES7 136-6BA00-0CA0  V1.0
      slot 1: "-K30006"  F-DI 8x24VDC HF
   slot 6: "-K30007"  F-DI 8x24VDC HF  6ES7 136-6BA00-0CA0  V1.0
      slot 1: "-K30007"  F-DI 8x24VDC HF
   slot 7: "-K30008"  F-DQ 4x24VDC/2A PM HF  6ES7 136-6DB00-0CA0  V2.0
      slot 1: "-K30008"  F-DQ 4x24VDC/2A PM HF
   slot 8: "-K30009"  F-DQ 4x24VDC/2A PM HF  6ES7 136-6DB00-0CA0  V2.0
      slot 1: "-K30009"  F-DQ 4x24VDC/2A PM HF
   slot 9: "-K30010"  F-DQ 4x24VDC/2A PM HF  6ES7 136-6DB00-0CA0  V2.0
      slot 1: "-K30010"  F-DQ 4x24VDC/2A PM HF
   slot 10: "-K30011"  F-DQ 4x24VDC/2A PM HF  6ES7 136-6DB00-0CA0  V2.0
      slot 1: "-K30011"  F-DQ 4x24VDC/2A PM HF
   slot 11: "-K30012"  F-DQ 4x24VDC/2A PM HF  6ES7 136-6DB00-0CA0  V2.0
      slot 1: "-K30012"  F-DQ 4x24VDC/2A PM HF
   slot 12: "-K30013"  F-DQ 4x24VDC/2A PM HF  6ES7 136-6DB00-0CA0  V2.0
      slot 1: "-K30013"  F-DQ 4x24VDC/2A PM HF
   slot 13: "Server module_1"  Server module  6ES7 193-6PA00-0AA0  V1.1
      slot 1: "Server module_1"  Server module
   slot 127: "BA 2xRJ45"  BA 2xRJ45  6ES7 193-6AR00-0AA0  V0.0
      slot 1: "Port_1"  X1 P1 R  6ES7 193-6AR00-0AA0  V0.0
      slot 2: "Port_2"  X1 P2 R  6ES7 193-6AR00-0AA0  V0.0
DEVICE "n0047-uc254-xn10"  GSD.Device.PN
   slot 0: "Rack"  Rack  V1.0
   slot 0: "n0047-uc254-xn10"  55556 MVK-MPNIO F DI16/8  55556
      slot 0: "55556 MVK-MPNIO F DI16/8_1"  55556 MVK-MPNIO F DI16/8
      slot 1: "55556 MVK-MPNIO F DI16/8"  55556 MVK-MPNIO F DI16/8
         slot 1: "Port 1"  Port 1
         slot 2: "Port 2"  Port 2
      slot 1: "Power module_1"  Power module
         slot 0: "Power module"  Power module
   slot 2: "-XN10"  FS Data
      slot 0: "-XN10"  FS Data
DEVICE "n0048-lv006-el001-k30001"  ET 200SP-Station
   slot 0: "Rack_0"  Rack  6ES5 710-8MAx1
   slot 0: "n0048-lv006-el001-k30001"  IM 155-6 PN ST  6ES7 155-6AU01-0BN0  V4.2
   slot 1: "-K30002"  DI 16x24VDC ST  6ES7 131-6BH01-0BA0  V0.0
      slot 1: "-K30002"  DI 16x24VDC ST
   slot 2: "-K30003"  F-DI 8x24VDC HF  6ES7 136-6BA00-0CA0  V1.0
      slot 1: "-K30003"  F-DI 8x24VDC HF
   slot 3: "-K30004"  F-DQ 4x24VDC/2A PM HF  6ES7 136-6DB00-0CA0  V2.0
      slot 1: "-K30004"  F-DQ 4x24VDC/2A PM HF
   slot 4: "Server module_1"  Server module  6ES7 193-6PA00-0AA0  V1.1
      slot 1: "Server module_1"  Server module
   slot 127: "BA 2xRJ45"  BA 2xRJ45  6ES7 193-6AR00-0AA0  V0.0
      slot 1: "Port_1"  X1 P1 R  6ES7 193-6AR00-0AA0  V0.0
      slot 2: "Port_2"  X1 P2 R  6ES7 193-6AR00-0AA0  V0.0
DEVICE "n0051-uc24-el001-k30001"  ET 200SP-Station
   slot 0: "Rack_0"  Rack  6ES5 710-8MAx1
   slot 0: "n0051-uc24-el001-k30001"  IM 155-6 PN ST  6ES7 155-6AU01-0BN0  V4.2
   slot 1: "-K30002"  DI 16x24VDC ST  6ES7 131-6BH01-0BA0  V0.0
      slot 1: "-K30002"  DI 16x24VDC ST
   slot 2: "-K30003"  DI 16x24VDC ST  6ES7 131-6BH01-0BA0  V0.0
      slot 1: "-K30003"  DI 16x24VDC ST
   slot 3: "-K30004"  F-DI 8x24VDC HF  6ES7 136-6BA00-0CA0  V1.0
      slot 1: "-K30004"  F-DI 8x24VDC HF
   slot 4: "-K30005"  F-DI 8x24VDC HF  6ES7 136-6BA00-0CA0  V1.0
      slot 1: "-K30005"  F-DI 8x24VDC HF
   slot 5: "-K30006"  F-DI 8x24VDC HF  6ES7 136-6BA00-0CA0  V1.0
      slot 1: "-K30006"  F-DI 8x24VDC HF
   slot 6: "-K30007"  F-DI 8x24VDC HF  6ES7 136-6BA00-0CA0  V1.0
      slot 1: "-K30007"  F-DI 8x24VDC HF
   slot 7: "-K30008"  F-DQ 4x24VDC/2A PM HF  6ES7 136-6DB00-0CA0  V2.0
      slot 1: "-K30008"  F-DQ 4x24VDC/2A PM HF
   slot 8: "-K30009"  F-DQ 4x24VDC/2A PM HF  6ES7 136-6DB00-0CA0  V2.0
      slot 1: "-K30009"  F-DQ 4x24VDC/2A PM HF
   slot 9: "-K30010"  F-DQ 4x24VDC/2A PM HF  6ES7 136-6DB00-0CA0  V2.0
      slot 1: "-K30010"  F-DQ 4x24VDC/2A PM HF
   slot 10: "-K30011"  F-DQ 4x24VDC/2A PM HF  6ES7 136-6DB00-0CA0  V2.0
      slot 1: "-K30011"  F-DQ 4x24VDC/2A PM HF
   slot 11: "-K30012"  F-DQ 4x24VDC/2A PM HF  6ES7 136-6DB00-0CA0  V2.0
      slot 1: "-K30012"  F-DQ 4x24VDC/2A PM HF
   slot 12: "-K30013"  F-DQ 4x24VDC/2A PM HF  6ES7 136-6DB00-0CA0  V2.0
      slot 1: "-K30013"  F-DQ 4x24VDC/2A PM HF
   slot 13: "Server module_1"  Server module  6ES7 193-6PA00-0AA0  V1.1
      slot 1: "Server module_1"  Server module
   slot 127: "BA 2xRJ45"  BA 2xRJ45  6ES7 193-6AR00-0AA0  V0.0
      slot 1: "Port_1"  X1 P1 R  6ES7 193-6AR00-0AA0  V0.0
      slot 2: "Port_2"  X1 P2 R  6ES7 193-6AR00-0AA0  V0.0
DEVICE "n0052-uc244-xn10"  GSD.Device.PN
   slot 0: "Rack"  Rack  V1.0
   slot 0: "n0052-uc244-xn10"  55556 MVK-MPNIO F DI16/8  55556
      slot 0: "55556 MVK-MPNIO F DI16/8_1"  55556 MVK-MPNIO F DI16/8
      slot 1: "55556 MVK-MPNIO F DI16/8"  55556 MVK-MPNIO F DI16/8
         slot 1: "Port 1"  Port 1
         slot 2: "Port 2"  Port 2
      slot 1: "Power module_1"  Power module
         slot 0: "Power module"  Power module
   slot 2: "-XN10"  FS Data
      slot 0: "-XN10"  FS Data
DEVICE "n0056-uc23-el001-k30001"  ET 200SP-Station
   slot 0: "Rack_0"  Rack  6ES5 710-8MAx1
   slot 0: "n0056-uc23-el001-k30001"  IM 155-6 PN ST  6ES7 155-6AU01-0BN0  V4.2
   slot 1: "-K30002"  DI 16x24VDC ST  6ES7 131-6BH01-0BA0  V0.0
      slot 1: "-K30002"  DI 16x24VDC ST
   slot 2: "-K30003"  DI 16x24VDC ST  6ES7 131-6BH01-0BA0  V0.0
      slot 1: "-K30003"  DI 16x24VDC ST
   slot 3: "-K30004"  F-DI 8x24VDC HF  6ES7 136-6BA00-0CA0  V1.0
      slot 1: "-K30004"  F-DI 8x24VDC HF
   slot 4: "-K30005"  F-DI 8x24VDC HF  6ES7 136-6BA00-0CA0  V1.0
      slot 1: "-K30005"  F-DI 8x24VDC HF
   slot 5: "-K30006"  F-DI 8x24VDC HF  6ES7 136-6BA00-0CA0  V1.0
      slot 1: "-K30006"  F-DI 8x24VDC HF
   slot 6: "-K30007"  F-DI 8x24VDC HF  6ES7 136-6BA00-0CA0  V1.0
      slot 1: "-K30007"  F-DI 8x24VDC HF
   slot 7: "-K30008"  F-DQ 4x24VDC/2A PM HF  6ES7 136-6DB00-0CA0  V2.0
      slot 1: "-K30008"  F-DQ 4x24VDC/2A PM HF
   slot 8: "-K30009"  F-DQ 4x24VDC/2A PM HF  6ES7 136-6DB00-0CA0  V2.0
      slot 1: "-K30009"  F-DQ 4x24VDC/2A PM HF
   slot 9: "-K30010"  F-DQ 4x24VDC/2A PM HF  6ES7 136-6DB00-0CA0  V2.0
      slot 1: "-K30010"  F-DQ 4x24VDC/2A PM HF
   slot 10: "-K30011"  F-DQ 4x24VDC/2A PM HF  6ES7 136-6DB00-0CA0  V2.0
      slot 1: "-K30011"  F-DQ 4x24VDC/2A PM HF
   slot 11: "-K30012"  F-DQ 4x24VDC/2A PM HF  6ES7 136-6DB00-0CA0  V2.0
      slot 1: "-K30012"  F-DQ 4x24VDC/2A PM HF
   slot 12: "-K30013"  F-DQ 4x24VDC/2A PM HF  6ES7 136-6DB00-0CA0  V2.0
      slot 1: "-K30013"  F-DQ 4x24VDC/2A PM HF
   slot 13: "Server module_1"  Server module  6ES7 193-6PA00-0AA0  V1.1
      slot 1: "Server module_1"  Server module
   slot 127: "BA 2xRJ45"  BA 2xRJ45  6ES7 193-6AR00-0AA0  V0.0
      slot 1: "Port_1"  X1 P1 R  6ES7 193-6AR00-0AA0  V0.0
      slot 2: "Port_2"  X1 P2 R  6ES7 193-6AR00-0AA0  V0.0
DEVICE "n0057-uc234-xn10"  GSD.Device.PN
   slot 0: "Rack"  Rack  V1.0
   slot 0: "n0057-uc234-xn10"  55556 MVK-MPNIO F DI16/8  55556
      slot 0: "55556 MVK-MPNIO F DI16/8_1"  55556 MVK-MPNIO F DI16/8
      slot 1: "55556 MVK-MPNIO F DI16/8"  55556 MVK-MPNIO F DI16/8
         slot 1: "Port 1"  Port 1
         slot 2: "Port 2"  Port 2
      slot 1: "Power module_1"  Power module
         slot 0: "Power module"  Power module
   slot 2: "-XN10"  FS Data
      slot 0: "-XN10"  FS Data
DEVICE "n0058-ct2-el003-k30001"  ET 200SP-Station
   slot 0: "Rack_0"  Rack  6ES5 710-8MAx1
   slot 0: "n0058-ct2-el003-k30001"  IM 155-6 PN ST  6ES7 155-6AU01-0BN0  V4.2
   slot 1: "-K30002"  DI 16x24VDC ST  6ES7 131-6BH01-0BA0  V0.0
      slot 1: "-K30002"  DI 16x24VDC ST
   slot 2: "-K30003"  F-DI 8x24VDC HF  6ES7 136-6BA00-0CA0  V1.0
      slot 1: "-K30003"  F-DI 8x24VDC HF
   slot 3: "-K30004"  F-DI 8x24VDC HF  6ES7 136-6BA00-0CA0  V1.0
      slot 1: "-K30004"  F-DI 8x24VDC HF
   slot 4: "-K30005"  F-DI 8x24VDC HF  6ES7 136-6BA00-0CA0  V1.0
      slot 1: "-K30005"  F-DI 8x24VDC HF
   slot 5: "-K30006"  F-DI 8x24VDC HF  6ES7 136-6BA00-0CA0  V1.0
      slot 1: "-K30006"  F-DI 8x24VDC HF
   slot 6: "-K30007"  F-DI 8x24VDC HF  6ES7 136-6BA00-0CA0  V1.0
      slot 1: "-K30007"  F-DI 8x24VDC HF
   slot 7: "-K30008"  F-DQ 4x24VDC/2A PM HF  6ES7 136-6DB00-0CA0  V2.0
      slot 1: "-K30008"  F-DQ 4x24VDC/2A PM HF
   slot 8: "-K30009"  F-DQ 4x24VDC/2A PM HF  6ES7 136-6DB00-0CA0  V2.0
      slot 1: "-K30009"  F-DQ 4x24VDC/2A PM HF
   slot 9: "Server module_1"  Server module  6ES7 193-6PA00-0AA0  V1.1
      slot 1: "Server module_1"  Server module
   slot 127: "BA 2xRJ45"  BA 2xRJ45  6ES7 193-6AR00-0AA0  V0.0
      slot 1: "Port_1"  X1 P1 R  6ES7 193-6AR00-0AA0  V0.0
      slot 2: "Port_2"  X1 P2 R  6ES7 193-6AR00-0AA0  V0.0
DEVICE "n0061-uc22-el001-k30001"  ET 200SP-Station
   slot 0: "Rack_0"  Rack  6ES5 710-8MAx1
   slot 0: "n0061-uc22-el001-k30001"  IM 155-6 PN ST  6ES7 155-6AU01-0BN0  V4.2
   slot 1: "-K30002"  DI 16x24VDC ST  6ES7 131-6BH01-0BA0  V0.0
      slot 1: "-K30002"  DI 16x24VDC ST
   slot 2: "-K30003"  DI 16x24VDC ST  6ES7 131-6BH01-0BA0  V0.0
      slot 1: "-K30003"  DI 16x24VDC ST
   slot 3: "-K30004"  F-DI 8x24VDC HF  6ES7 136-6BA00-0CA0  V1.0
      slot 1: "-K30004"  F-DI 8x24VDC HF
   slot 4: "-K30005"  F-DI 8x24VDC HF  6ES7 136-6BA00-0CA0  V1.0
      slot 1: "-K30005"  F-DI 8x24VDC HF
   slot 5: "-K30006"  F-DI 8x24VDC HF  6ES7 136-6BA00-0CA0  V1.0
      slot 1: "-K30006"  F-DI 8x24VDC HF
   slot 6: "-K30007"  F-DI 8x24VDC HF  6ES7 136-6BA00-0CA0  V1.0
      slot 1: "-K30007"  F-DI 8x24VDC HF
   slot 7: "-K30008"  F-DQ 4x24VDC/2A PM HF  6ES7 136-6DB00-0CA0  V2.0
      slot 1: "-K30008"  F-DQ 4x24VDC/2A PM HF
   slot 8: "-K30009"  F-DQ 4x24VDC/2A PM HF  6ES7 136-6DB00-0CA0  V2.0
      slot 1: "-K30009"  F-DQ 4x24VDC/2A PM HF
   slot 9: "-K30010"  F-DQ 4x24VDC/2A PM HF  6ES7 136-6DB00-0CA0  V2.0
      slot 1: "-K30010"  F-DQ 4x24VDC/2A PM HF
   slot 10: "-K30011"  F-DQ 4x24VDC/2A PM HF  6ES7 136-6DB00-0CA0  V2.0
      slot 1: "-K30011"  F-DQ 4x24VDC/2A PM HF
   slot 11: "-K30012"  F-DQ 4x24VDC/2A PM HF  6ES7 136-6DB00-0CA0  V2.0
      slot 1: "-K30012"  F-DQ 4x24VDC/2A PM HF
   slot 12: "-K30013"  F-DQ 4x24VDC/2A PM HF  6ES7 136-6DB00-0CA0  V2.0
      slot 1: "-K30013"  F-DQ 4x24VDC/2A PM HF
   slot 13: "Server module_1"  Server module  6ES7 193-6PA00-0AA0  V1.1
      slot 1: "Server module_1"  Server module
   slot 127: "BA 2xRJ45"  BA 2xRJ45  6ES7 193-6AR00-0AA0  V0.0
      slot 1: "Port_1"  X1 P1 R  6ES7 193-6AR00-0AA0  V0.0
      slot 2: "Port_2"  X1 P2 R  6ES7 193-6AR00-0AA0  V0.0
DEVICE "n0062-uc224-xn10"  GSD.Device.PN
   slot 0: "Rack"  Rack  V1.0
   slot 0: "n0062-uc224-xn10"  55556 MVK-MPNIO F DI16/8  55556
      slot 0: "55556 MVK-MPNIO F DI16/8_1"  55556 MVK-MPNIO F DI16/8
      slot 1: "55556 MVK-MPNIO F DI16/8"  55556 MVK-MPNIO F DI16/8
         slot 1: "Port 1"  Port 1
         slot 2: "Port 2"  Port 2
      slot 1: "Power module_1"  Power module
         slot 0: "Power module"  Power module
   slot 2: "-XN10"  FS Data
      slot 0: "-XN10"  FS Data
DEVICE "n0063-lv006-el001-k30001"  ET 200SP-Station
   slot 0: "Rack_0"  Rack  6ES5 710-8MAx1
   slot 0: "n0063-lv006-el001-k30001"  IM 155-6 PN ST  6ES7 155-6AU01-0BN0  V4.2
   slot 1: "-K30002"  DI 16x24VDC ST  6ES7 131-6BH01-0BA0  V0.0
      slot 1: "-K30002"  DI 16x24VDC ST
   slot 2: "-K30003"  F-DI 8x24VDC HF  6ES7 136-6BA00-0CA0  V1.0
      slot 1: "-K30003"  F-DI 8x24VDC HF
   slot 3: "-K30004"  F-DQ 4x24VDC/2A PM HF  6ES7 136-6DB00-0CA0  V2.0
      slot 1: "-K30004"  F-DQ 4x24VDC/2A PM HF
   slot 4: "Server module_1"  Server module  6ES7 193-6PA00-0AA0  V1.1
      slot 1: "Server module_1"  Server module
   slot 127: "BA 2xRJ45"  BA 2xRJ45  6ES7 193-6AR00-0AA0  V0.0
      slot 1: "Port_1"  X1 P1 R  6ES7 193-6AR00-0AA0  V0.0
      slot 2: "Port_2"  X1 P2 R  6ES7 193-6AR00-0AA0  V0.0
DEVICE "n0066-uc21-el001-k30001"  ET 200SP-Station
   slot 0: "Rack_0"  Rack  6ES5 710-8MAx1
   slot 0: "n0066-uc21-el001-k30001"  IM 155-6 PN ST  6ES7 155-6AU01-0BN0  V4.2
   slot 1: "-K30002"  DI 16x24VDC ST  6ES7 131-6BH01-0BA0  V0.0
      slot 1: "-K30002"  DI 16x24VDC ST
   slot 2: "-K30003"  DI 16x24VDC ST  6ES7 131-6BH01-0BA0  V0.0
      slot 1: "-K30003"  DI 16x24VDC ST
   slot 3: "-K30004"  F-DI 8x24VDC HF  6ES7 136-6BA00-0CA0  V1.0
      slot 1: "-K30004"  F-DI 8x24VDC HF
   slot 4: "-K30005"  F-DI 8x24VDC HF  6ES7 136-6BA00-0CA0  V1.0
      slot 1: "-K30005"  F-DI 8x24VDC HF
   slot 5: "-K30006"  F-DI 8x24VDC HF  6ES7 136-6BA00-0CA0  V1.0
      slot 1: "-K30006"  F-DI 8x24VDC HF
   slot 6: "-K30007"  F-DI 8x24VDC HF  6ES7 136-6BA00-0CA0  V1.0
      slot 1: "-K30007"  F-DI 8x24VDC HF
   slot 7: "-K30008"  F-DQ 4x24VDC/2A PM HF  6ES7 136-6DB00-0CA0  V2.0
      slot 1: "-K30008"  F-DQ 4x24VDC/2A PM HF
   slot 8: "-K30009"  F-DQ 4x24VDC/2A PM HF  6ES7 136-6DB00-0CA0  V2.0
      slot 1: "-K30009"  F-DQ 4x24VDC/2A PM HF
   slot 9: "-K30010"  F-DQ 4x24VDC/2A PM HF  6ES7 136-6DB00-0CA0  V2.0
      slot 1: "-K30010"  F-DQ 4x24VDC/2A PM HF
   slot 10: "-K30011"  F-DQ 4x24VDC/2A PM HF  6ES7 136-6DB00-0CA0  V2.0
      slot 1: "-K30011"  F-DQ 4x24VDC/2A PM HF
   slot 11: "-K30012"  F-DQ 4x24VDC/2A PM HF  6ES7 136-6DB00-0CA0  V2.0
      slot 1: "-K30012"  F-DQ 4x24VDC/2A PM HF
   slot 12: "-K30013"  F-DQ 4x24VDC/2A PM HF  6ES7 136-6DB00-0CA0  V2.0
      slot 1: "-K30013"  F-DQ 4x24VDC/2A PM HF
   slot 13: "Server module_1"  Server module  6ES7 193-6PA00-0AA0  V1.1
      slot 1: "Server module_1"  Server module
   slot 127: "BA 2xRJ45"  BA 2xRJ45  6ES7 193-6AR00-0AA0  V0.0
      slot 1: "Port_1"  X1 P1 R  6ES7 193-6AR00-0AA0  V0.0
      slot 2: "Port_2"  X1 P2 R  6ES7 193-6AR00-0AA0  V0.0
DEVICE "n0067-uc214-xn10"  GSD.Device.PN
   slot 0: "Rack"  Rack  V1.0
   slot 0: "n0067-uc214-xn10"  55556 MVK-MPNIO F DI16/8  55556
      slot 0: "55556 MVK-MPNIO F DI16/8_1"  55556 MVK-MPNIO F DI16/8
      slot 1: "55556 MVK-MPNIO F DI16/8"  55556 MVK-MPNIO F DI16/8
         slot 1: "Port 1"  Port 1
         slot 2: "Port 2"  Port 2
      slot 1: "Power module_1"  Power module
         slot 0: "Power module"  Power module
   slot 2: "-XN10"  FS Data
      slot 0: "-XN10"  FS Data
DEVICE "n0070-uf31-el001-k30001"  ET 200SP-Station
   slot 0: "Rack_0"  Rack  6ES5 710-8MAx1
   slot 0: "n0070-uf31-el001-k30001"  IM 155-6 PN ST  6ES7 155-6AU01-0BN0  V4.2
   slot 1: "-K30002"  DI 16x24VDC ST  6ES7 131-6BH01-0BA0  V0.0
      slot 1: "-K30002"  DI 16x24VDC ST
   slot 2: "-K30003"  F-DI 8x24VDC HF  6ES7 136-6BA00-0CA0  V1.0
      slot 1: "-K30003"  F-DI 8x24VDC HF
   slot 3: "-K30004"  F-DQ 4x24VDC/2A PM HF  6ES7 136-6DB00-0CA0  V2.0
      slot 1: "-K30004"  F-DQ 4x24VDC/2A PM HF
   slot 4: "-K30005"  F-DQ 4x24VDC/2A PM HF  6ES7 136-6DB00-0CA0  V2.0
      slot 1: "-K30005"  F-DQ 4x24VDC/2A PM HF
   slot 5: "Server module_1"  Server module  6ES7 193-6PA00-0AA0  V1.1
      slot 1: "Server module_1"  Server module
   slot 127: "BA 2xRJ45"  BA 2xRJ45  6ES7 193-6AR00-0AA0  V0.0
      slot 1: "Port_1"  X1 P1 R  6ES7 193-6AR00-0AA0  V0.0
      slot 2: "Port_2"  X1 P2 R  6ES7 193-6AR00-0AA0  V0.0
DEVICE "n0071-uf41-el001-k30001"  ET 200SP-Station
   slot 0: "Rack_0"  Rack  6ES5 710-8MAx1
   slot 0: "n0071-uf41-el001-k30001"  IM 155-6 PN ST  6ES7 155-6AU01-0BN0  V4.2
   slot 1: "-K30002"  DI 16x24VDC ST  6ES7 131-6BH01-0BA0  V0.0
      slot 1: "-K30002"  DI 16x24VDC ST
   slot 2: "-K30003"  F-DI 8x24VDC HF  6ES7 136-6BA00-0CA0  V1.0
      slot 1: "-K30003"  F-DI 8x24VDC HF
   slot 3: "-K30004"  F-DQ 4x24VDC/2A PM HF  6ES7 136-6DB00-0CA0  V2.0
      slot 1: "-K30004"  F-DQ 4x24VDC/2A PM HF
   slot 4: "-K30005"  F-DQ 4x24VDC/2A PM HF  6ES7 136-6DB00-0CA0  V2.0
      slot 1: "-K30005"  F-DQ 4x24VDC/2A PM HF
   slot 5: "Server module_1"  Server module  6ES7 193-6PA00-0AA0  V1.1
      slot 1: "Server module_1"  Server module
   slot 127: "BA 2xRJ45"  BA 2xRJ45  6ES7 193-6AR00-0AA0  V0.0
      slot 1: "Port_1"  X1 P1 R  6ES7 193-6AR00-0AA0  V0.0
      slot 2: "Port_2"  X1 P2 R  6ES7 193-6AR00-0AA0  V0.0
DEVICE "n0072-uf51-el001-k30001"  ET 200SP-Station
   slot 0: "Rack_0"  Rack  6ES5 710-8MAx1
   slot 0: "n0072-uf51-el001-k30001"  IM 155-6 PN ST  6ES7 155-6AU01-0BN0  V4.2
   slot 1: "-K30002"  DI 16x24VDC ST  6ES7 131-6BH01-0BA0  V0.0
      slot 1: "-K30002"  DI 16x24VDC ST
   slot 2: "-K30003"  F-DI 8x24VDC HF  6ES7 136-6BA00-0CA0  V1.0
      slot 1: "-K30003"  F-DI 8x24VDC HF
   slot 3: "-K30004"  F-DQ 4x24VDC/2A PM HF  6ES7 136-6DB00-0CA0  V2.0
      slot 1: "-K30004"  F-DQ 4x24VDC/2A PM HF
   slot 4: "-K30005"  F-DQ 4x24VDC/2A PM HF  6ES7 136-6DB00-0CA0  V2.0
      slot 1: "-K30005"  F-DQ 4x24VDC/2A PM HF
   slot 5: "Server module_1"  Server module  6ES7 193-6PA00-0AA0  V1.1
      slot 1: "Server module_1"  Server module
   slot 127: "BA 2xRJ45"  BA 2xRJ45  6ES7 193-6AR00-0AA0  V0.0
      slot 1: "Port_1"  X1 P1 R  6ES7 193-6AR00-0AA0  V0.0
      slot 2: "Port_2"  X1 P2 R  6ES7 193-6AR00-0AA0  V0.0
DEVICE "n0080-uf511-xn10"  GSD.Device.PN
   slot 0: "Rack"  Rack  V1.0
   slot 0: "n0080-uf511-xn10"  55556 MVK-MPNIO F DI16/8  55556
      slot 0: "55556 MVK-MPNIO F DI16/8_1"  55556 MVK-MPNIO F DI16/8
      slot 1: "55556 MVK-MPNIO F DI16/8"  55556 MVK-MPNIO F DI16/8
         slot 1: "Port 1"  Port 1
         slot 2: "Port 2"  Port 2
      slot 1: "Power module_1"  Power module
         slot 0: "Power module"  Power module
   slot 2: "-XN10"  FS Data
      slot 0: "-XN10"  FS Data
DEVICE "n0073-ifg31-el001-k30001"  ET 200SP-Station
   slot 0: "Rack_0"  Rack  6ES5 710-8MAx1
   slot 0: "n0073-ifg31-el001-k30001"  IM 155-6 PN ST  6ES7 155-6AU01-0BN0  V4.2
   slot 1: "-K30002"  DI 16x24VDC ST  6ES7 131-6BH01-0BA0  V0.0
      slot 1: "-K30002"  DI 16x24VDC ST
   slot 2: "-K30003"  F-DI 8x24VDC HF  6ES7 136-6BA00-0CA0  V1.0
      slot 1: "-K30003"  F-DI 8x24VDC HF
   slot 3: "-K30004"  F-DI 8x24VDC HF  6ES7 136-6BA00-0CA0  V1.0
      slot 1: "-K30004"  F-DI 8x24VDC HF
   slot 4: "-K30005"  F-DQ 4x24VDC/2A PM HF  6ES7 136-6DB00-0CA0  V2.0
      slot 1: "-K30005"  F-DQ 4x24VDC/2A PM HF
   slot 5: "-K30006"  F-DQ 4x24VDC/2A PM HF  6ES7 136-6DB00-0CA0  V2.0
      slot 1: "-K30006"  F-DQ 4x24VDC/2A PM HF
   slot 6: "Server module_1"  Server module  6ES7 193-6PA00-0AA0  V1.1
      slot 1: "Server module_1"  Server module
   slot 127: "BA 2xRJ45"  BA 2xRJ45  6ES7 193-6AR00-0AA0  V0.0
      slot 1: "Port_1"  X1 P1 R  6ES7 193-6AR00-0AA0  V0.0
      slot 2: "Port_2"  X1 P2 R  6ES7 193-6AR00-0AA0  V0.0
DEVICE "n0074-ifg41-el001-k30001"  ET 200SP-Station
   slot 0: "Rack_0"  Rack  6ES5 710-8MAx1
   slot 0: "n0074-ifg41-el001-k30001"  IM 155-6 PN ST  6ES7 155-6AU01-0BN0  V4.2
   slot 1: "-K30002"  DI 16x24VDC ST  6ES7 131-6BH01-0BA0  V0.0
      slot 1: "-K30002"  DI 16x24VDC ST
   slot 2: "-K30003"  F-DI 8x24VDC HF  6ES7 136-6BA00-0CA0  V1.0
      slot 1: "-K30003"  F-DI 8x24VDC HF
   slot 3: "-K30004"  F-DI 8x24VDC HF  6ES7 136-6BA00-0CA0  V1.0
      slot 1: "-K30004"  F-DI 8x24VDC HF
   slot 4: "-K30005"  F-DQ 4x24VDC/2A PM HF  6ES7 136-6DB00-0CA0  V2.0
      slot 1: "-K30005"  F-DQ 4x24VDC/2A PM HF
   slot 5: "-K30006"  F-DQ 4x24VDC/2A PM HF  6ES7 136-6DB00-0CA0  V2.0
      slot 1: "-K30006"  F-DQ 4x24VDC/2A PM HF
   slot 6: "Server module_1"  Server module  6ES7 193-6PA00-0AA0  V1.1
      slot 1: "Server module_1"  Server module
   slot 127: "BA 2xRJ45"  BA 2xRJ45  6ES7 193-6AR00-0AA0  V0.0
      slot 1: "Port_1"  X1 P1 R  6ES7 193-6AR00-0AA0  V0.0
      slot 2: "Port_2"  X1 P2 R  6ES7 193-6AR00-0AA0  V0.0
DEVICE "n0075-uf32-el001-k30001"  ET 200SP-Station
   slot 0: "Rack_0"  Rack  6ES5 710-8MAx1
   slot 0: "n0075-uf32-el001-k30001"  IM 155-6 PN ST  6ES7 155-6AU01-0BN0  V4.2
   slot 1: "-K30002"  DI 16x24VDC ST  6ES7 131-6BH01-0BA0  V0.0
      slot 1: "-K30002"  DI 16x24VDC ST
   slot 2: "-K30003"  F-DI 8x24VDC HF  6ES7 136-6BA00-0CA0  V1.0
      slot 1: "-K30003"  F-DI 8x24VDC HF
   slot 3: "-K30004"  F-DQ 4x24VDC/2A PM HF  6ES7 136-6DB00-0CA0  V2.0
      slot 1: "-K30004"  F-DQ 4x24VDC/2A PM HF
   slot 4: "-K30005"  F-DQ 4x24VDC/2A PM HF  6ES7 136-6DB00-0CA0  V2.0
      slot 1: "-K30005"  F-DQ 4x24VDC/2A PM HF
   slot 5: "-K30006"  F-DQ 4x24VDC/2A PM HF  6ES7 136-6DB00-0CA0  V2.0
      slot 1: "-K30006"  F-DQ 4x24VDC/2A PM HF
   slot 6: "Server module_1"  Server module  6ES7 193-6PA00-0AA0  V1.1
      slot 1: "Server module_1"  Server module
   slot 127: "BA 2xRJ45"  BA 2xRJ45  6ES7 193-6AR00-0AA0  V0.0
      slot 1: "Port_1"  X1 P1 R  6ES7 193-6AR00-0AA0  V0.0
      slot 2: "Port_2"  X1 P2 R  6ES7 193-6AR00-0AA0  V0.0
DEVICE "n0076-uf42-el001-k30001"  ET 200SP-Station
   slot 0: "Rack_0"  Rack  6ES5 710-8MAx1
   slot 0: "n0076-uf42-el001-k30001"  IM 155-6 PN ST  6ES7 155-6AU01-0BN0  V4.2
   slot 1: "-K30002"  DI 16x24VDC ST  6ES7 131-6BH01-0BA0  V0.0
      slot 1: "-K30002"  DI 16x24VDC ST
   slot 2: "-K30003"  F-DI 8x24VDC HF  6ES7 136-6BA00-0CA0  V1.0
      slot 1: "-K30003"  F-DI 8x24VDC HF
   slot 3: "-K30004"  F-DQ 4x24VDC/2A PM HF  6ES7 136-6DB00-0CA0  V2.0
      slot 1: "-K30004"  F-DQ 4x24VDC/2A PM HF
   slot 4: "-K30005"  F-DQ 4x24VDC/2A PM HF  6ES7 136-6DB00-0CA0  V2.0
      slot 1: "-K30005"  F-DQ 4x24VDC/2A PM HF
   slot 5: "Server module_1"  Server module  6ES7 193-6PA00-0AA0  V1.1
      slot 1: "Server module_1"  Server module
   slot 127: "BA 2xRJ45"  BA 2xRJ45  6ES7 193-6AR00-0AA0  V0.0
      slot 1: "Port_1"  X1 P1 R  6ES7 193-6AR00-0AA0  V0.0
      slot 2: "Port_2"  X1 P2 R  6ES7 193-6AR00-0AA0  V0.0
DEVICE "n0082-zp002-el001-k30001"  ET 200SP-Station
   slot 0: "Rack_0"  Rack  6ES5 710-8MAx1
   slot 0: "n0082-zp002-el001-k30001"  IM 155-6 PN ST  6ES7 155-6AU01-0BN0  V4.2
   slot 1: "-K30002"  DI 16x24VDC ST  6ES7 131-6BH01-0BA0  V0.0
      slot 1: "-K30002"  DI 16x24VDC ST
   slot 2: "-K30003"  F-DI 8x24VDC HF  6ES7 136-6BA00-0CA0  V1.0
      slot 1: "-K30003"  F-DI 8x24VDC HF
   slot 3: "-K30004"  F-DI 8x24VDC HF  6ES7 136-6BA00-0CA0  V1.0
      slot 1: "-K30004"  F-DI 8x24VDC HF
   slot 4: "-K30005"  F-DQ 4x24VDC/2A PM HF  6ES7 136-6DB00-0CA0  V2.0
      slot 1: "-K30005"  F-DQ 4x24VDC/2A PM HF
   slot 5: "-K30006"  DQ 16x24VDC/0.5A ST  6ES7 132-6BH01-0BA0  V0.0
      slot 1: "-K30006"  DQ 16x24VDC/0.5A ST
   slot 6: "Server module_1"  Server module  6ES7 193-6PA00-0AA0  V1.1
      slot 1: "Server module_1"  Server module
   slot 127: "BA 2xRJ45"  BA 2xRJ45  6ES7 193-6AR00-0AA0  V0.0
      slot 1: "Port_1"  X1 P1 R  6ES7 193-6AR00-0AA0  V0.0
      slot 2: "Port_2"  X1 P2 R  6ES7 193-6AR00-0AA0  V0.0
DEVICE "n0083-lv001-el001-k30001"  ET 200SP-Station
   slot 0: "Rack_0"  Rack  6ES5 710-8MAx1
   slot 0: "n0083-lv001-el001-k30001"  IM 155-6 PN ST  6ES7 155-6AU01-0BN0  V4.2
   slot 1: "-K30002"  DI 16x24VDC ST  6ES7 131-6BH01-0BA0  V0.0
      slot 1: "-K30002"  DI 16x24VDC ST
   slot 2: "-K30003"  F-DI 8x24VDC HF  6ES7 136-6BA00-0CA0  V1.0
      slot 1: "-K30003"  F-DI 8x24VDC HF
   slot 3: "-K30004"  F-DI 8x24VDC HF  6ES7 136-6BA00-0CA0  V1.0
      slot 1: "-K30004"  F-DI 8x24VDC HF
   slot 4: "-K30005"  F-DQ 4x24VDC/2A PM HF  6ES7 136-6DB00-0CA0  V2.0
      slot 1: "-K30005"  F-DQ 4x24VDC/2A PM HF
   slot 5: "-K30006"  F-DQ 4x24VDC/2A PM HF  6ES7 136-6DB00-0CA0  V2.0
      slot 1: "-K30006"  F-DQ 4x24VDC/2A PM HF
   slot 6: "Server module_1"  Server module  6ES7 193-6PA00-0AA0  V1.1
      slot 1: "Server module_1"  Server module
   slot 127: "BA 2xRJ45"  BA 2xRJ45  6ES7 193-6AR00-0AA0  V0.0
      slot 1: "Port_1"  X1 P1 R  6ES7 193-6AR00-0AA0  V0.0
      slot 2: "Port_2"  X1 P2 R  6ES7 193-6AR00-0AA0  V0.0
DEVICE "n0084-lv001-el001-k30001"  ET 200SP-Station
   slot 0: "Rack_0"  Rack  6ES5 710-8MAx1
   slot 0: "n0084-lv001-el001-k30001"  IM 155-6 PN ST  6ES7 155-6AU01-0BN0  V4.2
   slot 1: "-K30002"  DI 16x24VDC ST  6ES7 131-6BH01-0BA0  V0.0
      slot 1: "-K30002"  DI 16x24VDC ST
   slot 2: "-K30003"  F-DI 8x24VDC HF  6ES7 136-6BA00-0CA0  V1.0
      slot 1: "-K30003"  F-DI 8x24VDC HF
   slot 3: "-K30004"  F-DI 8x24VDC HF  6ES7 136-6BA00-0CA0  V1.0
      slot 1: "-K30004"  F-DI 8x24VDC HF
   slot 4: "-K30005"  F-DQ 4x24VDC/2A PM HF  6ES7 136-6DB00-0CA0  V2.0
      slot 1: "-K30005"  F-DQ 4x24VDC/2A PM HF
   slot 5: "-K30006"  F-DQ 4x24VDC/2A PM HF  6ES7 136-6DB00-0CA0  V2.0
      slot 1: "-K30006"  F-DQ 4x24VDC/2A PM HF
   slot 6: "Server module_1"  Server module  6ES7 193-6PA00-0AA0  V1.1
      slot 1: "Server module_1"  Server module
   slot 127: "BA 2xRJ45"  BA 2xRJ45  6ES7 193-6AR00-0AA0  V0.0
      slot 1: "Port_1"  X1 P1 R  6ES7 193-6AR00-0AA0  V0.0
      slot 2: "Port_2"  X1 P2 R  6ES7 193-6AR00-0AA0  V0.0
DEVICE "n0085-uc29-el001-k30001"  ET 200SP-Station
   slot 0: "Rack_0"  Rack  6ES5 710-8MAx1
   slot 0: "n0085-uc29-el001-k30001"  IM 155-6 PN ST  6ES7 155-6AU01-0BN0  V4.2
   slot 1: "-K30002"  DI 16x24VDC ST  6ES7 131-6BH01-0BA0  V0.0
      slot 1: "-K30002"  DI 16x24VDC ST
   slot 2: "-K30003"  F-DI 8x24VDC HF  6ES7 136-6BA00-0CA0  V1.0
      slot 1: "-K30003"  F-DI 8x24VDC HF
   slot 3: "-K30004"  F-DI 8x24VDC HF  6ES7 136-6BA00-0CA0  V1.0
      slot 1: "-K30004"  F-DI 8x24VDC HF
   slot 4: "-K30005"  F-DI 8x24VDC HF  6ES7 136-6BA00-0CA0  V1.0
      slot 1: "-K30005"  F-DI 8x24VDC HF
   slot 5: "-K30006"  F-DQ 4x24VDC/2A PM HF  6ES7 136-6DB00-0CA0  V2.0
      slot 1: "-K30006"  F-DQ 4x24VDC/2A PM HF
   slot 6: "Server module_1"  Server module  6ES7 193-6PA00-0AA0  V1.1
      slot 1: "Server module_1"  Server module
   slot 127: "BA 2xRJ45"  BA 2xRJ45  6ES7 193-6AR00-0AA0  V0.0
      slot 1: "Port_1"  X1 P1 R  6ES7 193-6AR00-0AA0  V0.0
      slot 2: "Port_2"  X1 P2 R  6ES7 193-6AR00-0AA0  V0.0
DEVICE "n0092-zp001-el001-k24501"  PnPn.Device
   slot 0: "Rack"  Rail  1.0
   slot 0: "n0092-zp001-el001-k24501"  PN/PN Coupler  6ES7 158-3AD10-0XA0  V4.2
   slot 1: "UNDEFINED_4"  PN/PN Coupler  6ES7 158-3AD10-0XA0  V4.2
   slot 127: "BA 2xRJ45"  BA 2xRJ45  6ES7 193-6AR00-0AA0  V0.0
      slot 1: "Port_1"  X1 P1 R  6ES7 193-6AR00-0AA0  V0.0
      slot 2: "Port_2"  X1 P2 R  6ES7 193-6AR00-0AA0  V0.0
   slot 127: "BA 2xRJ45"  BA 2xRJ45  6ES7 193-6AR00-0AA0  V0.0
      slot 1: "Port_1"  X2 P1 R  6ES7 193-6AR00-0AA0  V0.0
      slot 2: "Port_2"  X2 P2 R  6ES7 193-6AR00-0AA0  V0.0
DEVICE "n0091-zp001-el001-k30001"  ET 200SP-Station
   slot 0: "Rack_0"  Rack  6ES5 710-8MAx1
   slot 0: "n0091-zp001-el001-k30001"  IM 155-6 PN ST  6ES7 155-6AU01-0BN0  V4.2
   slot 1: "-K40002"  DI 16x24VDC ST  6ES7 131-6BH01-0BA0  V0.0
      slot 1: "-K40002"  DI 16x24VDC ST
   slot 2: "-K40003"  F-DI 8x24VDC HF  6ES7 136-6BA00-0CA0  V1.0
      slot 1: "-K40003"  F-DI 8x24VDC HF
   slot 3: "-K40004"  F-DI 8x24VDC HF  6ES7 136-6BA00-0CA0  V1.0
      slot 1: "-K40004"  F-DI 8x24VDC HF
   slot 4: "-K40005"  F-DI 8x24VDC HF  6ES7 136-6BA00-0CA0  V1.0
      slot 1: "-K40005"  F-DI 8x24VDC HF
   slot 5: "-K40010"  F-DI 8x24VDC HF  6ES7 136-6BA00-0CA0  V1.0
      slot 1: "-K40010"  F-DI 8x24VDC HF
   slot 6: "-K40006"  F-DQ 4x24VDC/2A PM HF  6ES7 136-6DB00-0CA0  V2.0
      slot 1: "-K40006"  F-DQ 4x24VDC/2A PM HF
   slot 7: "-K40007"  F-DQ 4x24VDC/2A PM HF  6ES7 136-6DB00-0CA0  V2.0
      slot 1: "-K40007"  F-DQ 4x24VDC/2A PM HF
   slot 8: "-K40008"  F-DQ 4x24VDC/2A PM HF  6ES7 136-6DB00-0CA0  V2.0
      slot 1: "-K40008"  F-DQ 4x24VDC/2A PM HF
   slot 9: "-K40009"  DQ 16x24VDC/0.5A ST  6ES7 132-6BH01-0BA0  V0.0
      slot 1: "-K40009"  DQ 16x24VDC/0.5A ST
   slot 10: "Server module_1"  Server module  6ES7 193-6PA00-0AA0  V1.1
      slot 1: "Server module_1"  Server module
   slot 127: "BA 2xRJ45"  BA 2xRJ45  6ES7 193-6AR00-0AA0  V0.0
      slot 1: "Port_1"  X1 P1 R  6ES7 193-6AR00-0AA0  V0.0
      slot 2: "Port_2"  X1 P2 R  6ES7 193-6AR00-0AA0  V0.0
DEVICE "n0093-ug7-el001-k30001"  ET 200SP-Station
   slot 0: "Rack_0"  Rack  6ES5 710-8MAx1
   slot 0: "n0093-ug7-el001-k30001"  IM 155-6 PN ST  6ES7 155-6AU01-0BN0  V4.2
   slot 1: "-K30002"  DI 16x24VDC ST  6ES7 131-6BH01-0BA0  V0.0
      slot 1: "-K30002"  DI 16x24VDC ST
   slot 2: "-K30003"  DI 16x24VDC ST  6ES7 131-6BH01-0BA0  V0.0
      slot 1: "-K30003"  DI 16x24VDC ST
   slot 3: "-K30004"  F-DI 8x24VDC HF  6ES7 136-6BA00-0CA0  V1.0
      slot 1: "-K30004"  F-DI 8x24VDC HF
   slot 4: "-K30005"  F-DI 8x24VDC HF  6ES7 136-6BA00-0CA0  V1.0
      slot 1: "-K30005"  F-DI 8x24VDC HF
   slot 5: "-K30006"  F-DI 8x24VDC HF  6ES7 136-6BA00-0CA0  V1.0
      slot 1: "-K30006"  F-DI 8x24VDC HF
   slot 6: "-K30007"  F-DI 8x24VDC HF  6ES7 136-6BA00-0CA0  V1.0
      slot 1: "-K30007"  F-DI 8x24VDC HF
   slot 7: "-K30008"  F-DQ 4x24VDC/2A PM HF  6ES7 136-6DB00-0CA0  V2.0
      slot 1: "-K30008"  F-DQ 4x24VDC/2A PM HF
   slot 8: "-K30009"  F-DQ 4x24VDC/2A PM HF  6ES7 136-6DB00-0CA0  V2.0
      slot 1: "-K30009"  F-DQ 4x24VDC/2A PM HF
   slot 9: "-K30010"  F-DQ 4x24VDC/2A PM HF  6ES7 136-6DB00-0CA0  V2.0
      slot 1: "-K30010"  F-DQ 4x24VDC/2A PM HF
   slot 10: "-K30011"  F-DQ 4x24VDC/2A PM HF  6ES7 136-6DB00-0CA0  V2.0
      slot 1: "-K30011"  F-DQ 4x24VDC/2A PM HF
   slot 11: "-K30012"  F-DQ 4x24VDC/2A PM HF  6ES7 136-6DB00-0CA0  V2.0
      slot 1: "-K30012"  F-DQ 4x24VDC/2A PM HF
   slot 12: "-K30013"  F-DQ 4x24VDC/2A PM HF  6ES7 136-6DB00-0CA0  V2.0
      slot 1: "-K30013"  F-DQ 4x24VDC/2A PM HF
   slot 13: "-K30014"  F-DQ 4x24VDC/2A PM HF  6ES7 136-6DB00-0CA0  V2.0
      slot 1: "-K30014"  F-DQ 4x24VDC/2A PM HF
   slot 14: "Server module_1"  Server module  6ES7 193-6PA00-0AA0  V1.1
      slot 1: "Server module_1"  Server module
   slot 127: "BA 2xRJ45"  BA 2xRJ45  6ES7 193-6AR00-0AA0  V0.0
      slot 1: "Port_1"  X1 P1 R  6ES7 193-6AR00-0AA0  V0.0
      slot 2: "Port_2"  X1 P2 R  6ES7 193-6AR00-0AA0  V0.0
DEVICE "n0094-ug7-xn10"  GSD.Device.PN
   slot 0: "Rack"  Rack  V1.0
   slot 0: "n0094-ug7-xn10"  55556 MVK-MPNIO F DI16/8  55556
      slot 0: "55556 MVK-MPNIO F DI16/8_1"  55556 MVK-MPNIO F DI16/8
      slot 1: "55556 MVK-MPNIO F DI16/8"  55556 MVK-MPNIO F DI16/8
         slot 1: "Port 1"  Port 1
         slot 2: "Port 2"  Port 2
      slot 1: "Power module_1"  Power module
         slot 0: "Power module"  Power module
   slot 2: "-XN10"  FS Data
      slot 0: "-XN10"  FS Data
*)

// ===== PLC "n0001-zp001-el001-k30001"  CPU 1517F-3 PN/DP =====
// protected blocks, not shown: "PNDD_IL_Diag_V1_11"

VAR_GLOBAL   // PLC tag table "Default tag table_1"
   "Tag_1" AT %Q10002.0 : Bool;
   "Tag_2" AT %Q100.0 : Bool;
   "System_Byte" AT %MB1 : Byte;
   "FirstScan" AT %M1.0 : Bool;
   "DiagStatusUpdate" AT %M1.1 : Bool;
   "AlwaysTRUE" AT %M1.2 : Bool;
   "AlwaysFALSE" AT %M1.3 : Bool;
   "Clock_Byte" AT %MB0 : Byte;
   "Clock_10Hz" AT %M0.0 : Bool;
   "Clock_5Hz" AT %M0.1 : Bool;
   "Clock_2.5Hz" AT %M0.2 : Bool;
   "Clock_2Hz" AT %M0.3 : Bool;
   "Clock_1.25Hz" AT %M0.4 : Bool;
   "Clock_1Hz" AT %M0.5 : Bool;
   "Clock_0.625Hz" AT %M0.6 : Bool;
   "Clock_0.5Hz" AT %M0.7 : Bool;
   "Tag_3" AT %Q0.0 : Bool;
   "Tag_4" AT %Q10002.1 : Bool;
   "Tag_5" AT %Q10002.2 : Bool;
   "Tag_6" AT %Q10005.0 : Bool;
   "ACKNOWLEDGE_PROGRAM_ALARMS" AT %M2.0 : Bool;
END_VAR

VAR_GLOBAL CONSTANT   // PLC tag table "Default tag table_1"
   "None(1)" : Pip := 65535;
   "Automatic update(1)" : Pip := 0;
   "PIP 1(1)" : Pip := 1;
   "PIP 2(1)" : Pip := 2;
   "PIP 3(1)" : Pip := 3;
   "PIP 4(1)" : Pip := 4;
   "PIP 5(1)" : Pip := 5;
   "PIP 6(1)" : Pip := 6;
   "PIP 7(1)" : Pip := 7;
   "PIP 8(1)" : Pip := 8;
   "PIP 9(1)" : Pip := 9;
   "PIP 10(1)" : Pip := 10;
   "PIP 11(1)" : Pip := 11;
   "PIP 12(1)" : Pip := 12;
   "PIP 13(1)" : Pip := 13;
   "PIP 14(1)" : Pip := 14;
   "PIP 15(1)" : Pip := 15;
   "PIP 16(1)" : Pip := 16;
   "PIP 17(1)" : Pip := 17;
   "PIP 18(1)" : Pip := 18;
   "PIP 19(1)" : Pip := 19;
   "PIP 20(1)" : Pip := 20;
   "PIP 21(1)" : Pip := 21;
   "PIP 22(1)" : Pip := 22;
   "PIP 23(1)" : Pip := 23;
   "PIP 24(1)" : Pip := 24;
   "PIP 25(1)" : Pip := 25;
   "PIP 26(1)" : Pip := 26;
   "PIP 27(1)" : Pip := 27;
   "PIP 28(1)" : Pip := 28;
   "PIP 29(1)" : Pip := 29;
   "PIP 30(1)" : Pip := 30;
   "PIP 31(1)" : Pip := 31;
   "PIP OB Servo(1)" : Pip := 32768;
   "Local~MC(1)" : Hw_SubModule := 51;
   "Local~Display(1)" : Hw_SubModule := 54;
   "Local~Exec(1)" : Hw_SubModule := 52;
   "Local(1)" : Hw_SubModule := 49;
   "Local~FExec(1)" : Hw_SubModule := 55;
   "Local~PROFINET_interface_1(1)" : Hw_Interface := 64;
   "Local~PROFINET_interface_1~Port_1(1)" : Hw_Interface := 65;
   "Local~PROFINET_interface_1~Port_2(1)" : Hw_Interface := 66;
   "Local~PROFINET_interface_2(1)" : Hw_Interface := 72;
   "Local~PROFINET_interface_2~Port_1(1)" : Hw_Interface := 73;
   "Local~Virtual_communication_interface(1)" : Hw_Interface := 135;
   "OB_Main(1)" : OB_PCYCLE := 1;
   "OB_FOB_RTG1(1)" : OB_Cyclic := 123;
   "OB_IO access error" : OB_Any := 122;
   "OB_Programming error" : OB_Any := 121;
   "OB_FOB_RTG2" : OB_Cyclic := 124;
   "Local~PROFINET_IO-System" : Hw_IoSystem := 257;
   "Local~PROFINET_IO-System_1" : Hw_IoSystem := 258;
   "Local~Common(1)" : Hw_SubModule := 50;
   "Local~Device(1)" : Hw_Device := 32;
   "Local~Configuration(1)" : Hw_SubModule := 33;
   "Local~License_Manager(1)" : Hw_SubModule := 42;
   "Local~DP_interface_1(1)" : Hw_Interface := 60;
   "Local~n0001-zp001-el001-k30002(1)" : Hw_SubModule := 260;
   "Local~n0001-zp001-el001-k30002~PROFINET_interface_1(1)" : Hw_Interface := 261;
   "Local~n0001-zp001-el001-k30002~PROFINET_interface_1~Port_1(1)" : Hw_Interface := 262;
   "Local~n0001-zp001-el001-k30002~PROFINET_interface_1~Port_2(1)" : Hw_Interface := 263;
END_VAR

